// TIA Portal project "电厂_干燥机_V14" (V14)

(* hardware
DEVICE "S7-1200 station_1"  S7-1200 Station
   slot 0: "Rack_0"  Rack  V1.0
   slot 1: "PLC_1"  CPU 1214C AC/DC/Rly  6ES7 214-1BG40-0XB0  V4.2
   slot 101: "CM 1242-5"  CM 1242-5  6GK7 242-5DX30-0XE0  V1.0
DEVICE "HMI_2"  KTP700 Basic PN
   slot 0: "KTP700 Basic PN"  KTP700 Basic PN  6AV2 123-2GB03-0AX0  14.0.0.0
   slot 1: "HMI_RT_2"  KTP700 Basic PN  6AV2 123-2GB03-0AX0  14.0.0.0
   slot 5: "HMI_2.IE_CP_1"  PROFINET Interface  14.0.0.0
      slot 1: "PROFINET Interface_1"  PROFINET Interface
         slot 1: "Port_1"  Port
*)

// ===== PLC "PLC_1"  CPU 1214C AC/DC/Rly =====

VAR_GLOBAL   // PLC tag table "默认变量表"
   "System_Byte" AT %MB1 : Byte;
   "FirstScan" AT %M1.0 : Bool;
   "DiagStatusUpdate" AT %M1.1 : Bool;
   "AlwaysTRUE" AT %M1.2 : Bool;
   "AlwaysFALSE" AT %M1.3 : Bool;
   "Clock_Byte" AT %MB0 : Byte;
   "BClock_10Hz" AT %M0.0 : Bool;
   "Clock_5Hz" AT %M0.1 : Bool;
   "Clock_2.5Hz" AT %M0.2 : Bool;
   "Clock_2Hz" AT %M0.3 : Bool;
   "Clock_1.25Hz" AT %M0.4 : Bool;
   "Clock_1Hz" AT %M0.5 : Bool;
   "Clock_0.625Hz" AT %M0.6 : Bool;
   "Clock_0.5Hz" AT %M0.7 : Bool;
   "MB_COMM_LOAD_DONE" AT %M1.4 : Bool;
   "MB_COMM_LOAD_ERROR" AT %M1.5 : Bool;
   "MB_COMM_LOAD_STATUS" AT %MW1 : UInt;
   "MB_SLAVE_EN" AT %M1.6 : Bool;
END_VAR

VAR_GLOBAL   // PLC tag table "IO"
   "露点温度" AT %IW64 : Int;
   "加热温度" AT %IW66 : Int;
   "开机" AT %I0.0 : Bool;
   "停机" AT %I0.1 : Bool;
   "本地远程转换" AT %I0.2 : Bool;
   "远程开机" AT %I0.3 : Bool;
   "远程停机" AT %I0.4 : Bool;
   "进气低压" AT %I0.6 : Bool;
   "A塔进气阀" AT %Q0.0 : Bool;
   "B塔进气阀" AT %Q0.1 : Bool;
   "A塔排气阀" AT %Q0.2 : Bool;
   "B塔排气阀" AT %Q0.3 : Bool;
   "主加热" AT %Q0.4 : Bool;
   "辅加热" AT %Q0.5 : Bool;
   "运行指示" AT %Q0.6 : Bool;
   "故障指示" AT %Q0.7 : Bool;
   "远程指示" AT %Q1.0 : Bool;
END_VAR

// folder: IO

DATA_BLOCK "AI_conversion_DB"   // DB5
{ S7_Optimized_Access := 'TRUE' }
VERSION : 0.1
// stored: InstanceOfName ai_conversion
"ai_conversion"
BEGIN
END_DATA_BLOCK

// folder: Logic

DATA_BLOCK "PARAM_CONFIG_DB"   // DB6
{ S7_Optimized_Access := 'TRUE' }
VERSION : 0.1
// stored: InstanceOfName PARAM_Config
"PARAM_Config"
BEGIN
END_DATA_BLOCK

DATA_BLOCK "CTR_CYCLIC_DB"   // DB7
{ S7_Optimized_Access := 'TRUE' }
VERSION : 0.1
// stored: InstanceOfName CTR_Cyclic
"CTR_Cyclic"
BEGIN
END_DATA_BLOCK

DATA_BLOCK "AlarmError_DB"   // DB8
{ S7_Optimized_Access := 'TRUE' }
VERSION : 0.1
// stored: InstanceOfName Alarm_Error
"Alarm_Error"
BEGIN
END_DATA_BLOCK

// folder: ModbusRTU

DATA_BLOCK "mb_hold_reg"   // DB3
{ S7_Optimized_Access := 'FALSE' }
VERSION : 0.1
   VAR
      hold_registers : Array[0..99] of UInt;
   END_VAR
BEGIN
END_DATA_BLOCK

DATA_BLOCK "modbusrtu_DB"   // DB4
{ S7_Optimized_Access := 'TRUE' }
VERSION : 0.1
// stored: InstanceOfName modbusrtu
"modbusrtu"
BEGIN
END_DATA_BLOCK

// folder: (top level)

ORGANIZATION_BLOCK "Main"   // OB1, LAD, ProgramCycle
TITLE = "Main Program Sweep (Cycle)"
{ S7_Optimized_Access := 'TRUE' }
VERSION : 0.1
   VAR_TEMP   // added for the SCL form of the ladder/FBD networks
      _w1 : Bool;
   END_VAR
BEGIN

REGION Network 1: PARAM_Config
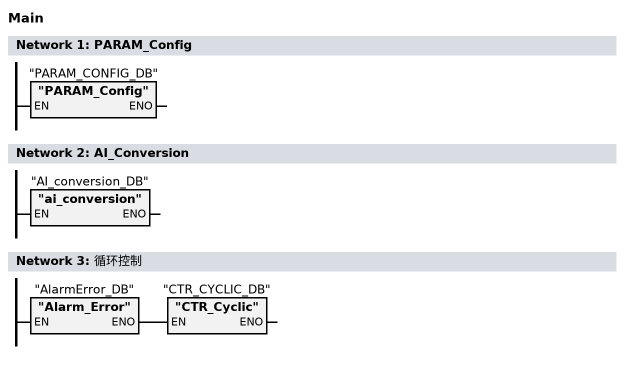
   RUNG wire#powerrail
      "PARAM_CONFIG_DB"()
   END_RUNG
   // the same network as SCL:
   "PARAM_CONFIG_DB"();   // "PARAM_Config"
END_REGION

REGION Network 2: AI_Conversion
   RUNG wire#powerrail
      "AI_conversion_DB"()
   END_RUNG
   // the same network as SCL:
   "AI_conversion_DB"();   // "ai_conversion"
END_REGION

REGION Network 3: 循环控制
   RUNG wire#powerrail
      "AlarmError_DB"()
      "CTR_CYCLIC_DB"()
   END_RUNG
   // the same network as SCL:
   "AlarmError_DB"(ENO => #_w1);   // "Alarm_Error"
   IF #_w1 THEN
       "CTR_CYCLIC_DB"();   // "CTR_Cyclic"
   END_IF;
END_REGION
END_ORGANIZATION_BLOCK

ORGANIZATION_BLOCK "Startup"   // OB100, LAD, Startup
TITLE = "Complete Restart"
{ S7_Optimized_Access := 'TRUE' }
VERSION : 0.1
   VAR_INPUT
      LostRetentive : Bool;   // True if retentive data are lost
      LostRTC : Bool;   // True if date and time are lost
   END_VAR
BEGIN

REGION Network 1: 运行时间计时初始化
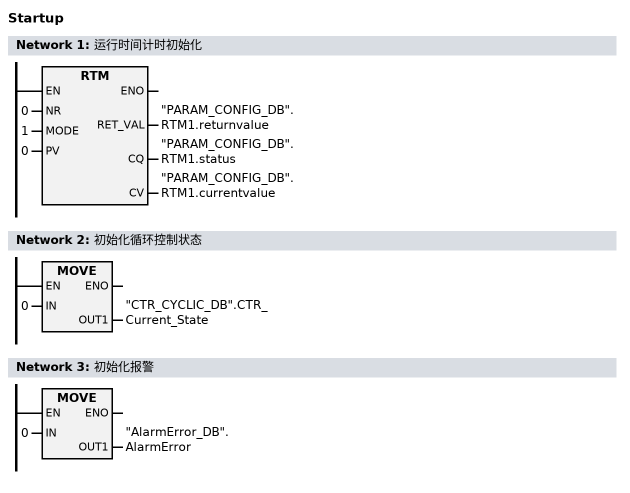
   "PARAM_CONFIG_DB".RTM1.returnvalue := RTM(NR := 0,
                           MODE := 1,
                           PV := 0,
                           CQ => "PARAM_CONFIG_DB".RTM1.status,
                           CV => "PARAM_CONFIG_DB".RTM1.currentvalue);
END_REGION

REGION Network 2: 初始化循环控制状态
   RUNG wire#powerrail
      Move(in := 0, out1 => "CTR_CYCLIC_DB".CTR_Current_State)
   END_RUNG
   // the same network as SCL:
   "CTR_CYCLIC_DB".CTR_Current_State := 0;
END_REGION

REGION Network 3: 初始化报警
   RUNG wire#powerrail
      Move(in := 0, out1 => "AlarmError_DB".AlarmError)
   END_RUNG
   // the same network as SCL:
   "AlarmError_DB".AlarmError := 0;
END_REGION
END_ORGANIZATION_BLOCK

// folder: IO

FUNCTION_BLOCK "ai_conversion"   // FB2, LAD
{ S7_Optimized_Access := 'TRUE' }
VERSION : 0.1
   VAR
      露点温度ac : Real;
      加热温度ac : Real;
   END_VAR
BEGIN

REGION Network 1: 露点温度线性变换
   // 露点温度传感器范围:-80-20摄氏度
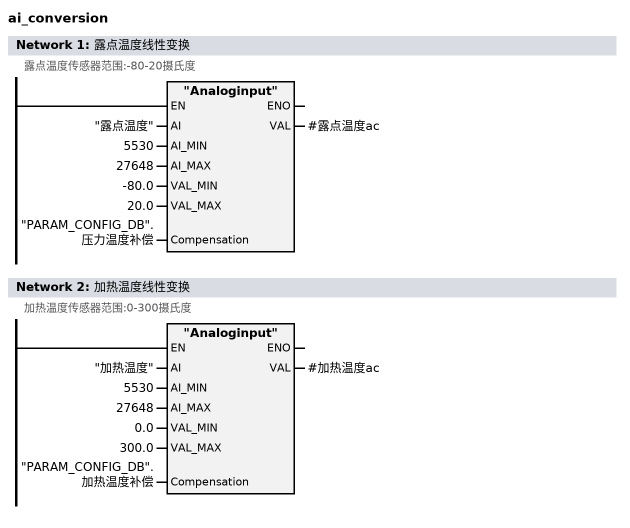
   RUNG wire#powerrail
      "Analoginput"(AI := "露点温度", AI_MIN := 5530, AI_MAX := 27648, VAL_MIN := -80.0, VAL_MAX := 20.0, Compensation := "PARAM_CONFIG_DB".压力温度补偿, VAL => #露点温度ac)
   END_RUNG
   // the same network as SCL:
   "Analoginput"(AI := "露点温度",
                 AI_MIN := 5530,
                 AI_MAX := 27648,
                 VAL_MIN := -80.0,
                 VAL_MAX := 20.0,
                 Compensation := "PARAM_CONFIG_DB".压力温度补偿,
                 VAL => #露点温度ac);
END_REGION

REGION Network 2: 加热温度线性变换
   // 加热温度传感器范围:0-300摄氏度
   RUNG wire#powerrail
      "Analoginput"(AI := "加热温度", AI_MIN := 5530, AI_MAX := 27648, VAL_MIN := 0.0, VAL_MAX := 300.0, Compensation := "PARAM_CONFIG_DB".加热温度补偿, VAL => #加热温度ac)
   END_RUNG
   // the same network as SCL:
   "Analoginput"(AI := "加热温度",
                 AI_MIN := 5530,
                 AI_MAX := 27648,
                 VAL_MIN := 0.0,
                 VAL_MAX := 300.0,
                 Compensation := "PARAM_CONFIG_DB".加热温度补偿,
                 VAL => #加热温度ac);
END_REGION
END_FUNCTION_BLOCK

FUNCTION "Analoginput" : Void   // FC71, LAD
TITLE = 模拟输入量处理
{ S7_Optimized_Access := 'TRUE' }
VERSION : 0.1
   VAR_INPUT
      AI : Int;   // 待处理模拟量
      AI_MIN : Int;   // 模拟量下限值
      AI_MAX : Int;   // 模拟量上限值
      VAL_MIN : Real;   // 实际值下限值
      VAL_MAX : Real;   // 实际值上限值
      Compensation : Real;
   END_VAR
   VAR_OUTPUT
      VAL : Real;   // 转换后的值
   END_VAR
   VAR_TEMP
      NORM_Out : Real;   // 模拟标准量
      SCALE_Out : Real;
   END_VAR
BEGIN

REGION Network 1: 标准化和缩放输入模拟量
   // 如果输入大于0,进行线性变换,否则赋值为0. / 输入模拟量是负值时,置零;
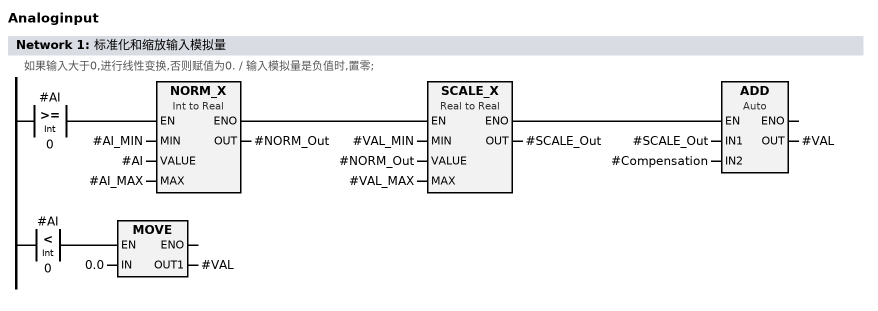
   RUNG wire#powerrail
      { S7_Templates := "SrcType := Int" } GE_Contact(in1 := #AI, in2 := 0)
      { S7_Templates := "[SrcType := Int, DestType := Real]"; S7_GenerateENO := "TRUE" } Normalize(min := #AI_MIN, value := #AI, max := #AI_MAX, out => #NORM_Out)
      { S7_Templates := "[SrcType := Real, DestType := Real]"; S7_GenerateENO := "TRUE" } Scale(min := #VAL_MIN, value := #NORM_Out, max := #VAL_MAX, out => #SCALE_Out)
      Add(in1 := #SCALE_Out, in2 := #Compensation, out => #VAL)
   END_RUNG
   RUNG wire#powerrail
      { S7_Templates := "SrcType := Int" } LT_Contact(in1 := #AI, in2 := 0)
      { S7_GenerateENO := "TRUE" } Move(in := 0.0, out1 => #VAL)
   END_RUNG
   // the same network as SCL:
   // ENO of a box is taken as its EN; it also drops when the box reports an error
   IF #AI >= 0 THEN
       #NORM_Out := NORM_X(MIN := #AI_MIN, VALUE := #AI, MAX := #AI_MAX);
       #SCALE_Out := SCALE_X(MIN := #VAL_MIN, VALUE := #NORM_Out, MAX := #VAL_MAX);
       #VAL := #SCALE_Out + #Compensation;
   END_IF;
   IF #AI < 0 THEN #VAL := 0.0; END_IF;
END_REGION
END_FUNCTION

// folder: Logic

FUNCTION_BLOCK "PARAM_Config"   // FB3, LAD
{ S7_Optimized_Access := 'TRUE' }
VERSION : 0.1
   VAR RETAIN
      主加热温度上限 : UInt := 120;   // 0～300℃
      主加热温度下限 : UInt := 100;   // 0～300℃
      加热超限温度报警 : UInt := 180;   // 0～300℃
      露点超限温度 : Int := -10;   // -500℃～500℃
      加热温度补偿 : Int := 0;   // -500℃～500℃
      压力温度补偿 : Int := 0;   // -500℃～500℃
      工作露点设定 : Int := -30;   // -500℃～500℃
      停机充压时间 : UDInt := 60;   // 3～999秒
      A塔工作B塔待再生 : UDInt := 10;   // 0～3600秒
      A塔工作B塔热再生 : UDInt := 25;   // 0～3600分
      A塔工作B塔吹冷 : UDInt := 15;   // 0～3600分
      A塔工作B塔充压 : UDInt := 8;   // 0～3600分
      A塔B塔均压 : UDInt := 10;   // 0～3600秒
      故障判断延时 : UInt := 5;   // 0～3600秒
      保养时间设定 : UDInt := 0;   // 0～100000h
      从站地址 : UInt := 2;   // 1～255
      露点控制最长延时 : UInt := 60;   // 0～3600分
   END_VAR
   VAR
      BT_Function : Struct
         BT_Runtime_Reset : Bool;
         BT_RuntimeReset_PREStatus : Bool;
      END_STRUCT;
      IEC_Timer_0_Instance : TONR_TIME;
      RTM1 : Struct
         returnvalue : Int;
         status : Bool;
         currentvalue : DInt;
         mode : UInt;
      END_STRUCT;
      MaintainTime_CountdownValue : Real;
   END_VAR
   VAR CONSTANT
      主加热温度上限_default : UInt := 120;   // default
      主加热温度下限_default : UInt := 100;   // default
      加热超限温度报警_default : UInt := 180;   // default
      露点超限温度_default : Int := -10;   // default
      加热温度补偿_default : Int := 0;   // default
      露点温度补偿_default : Int := 0;   // default
      工作露点设定_default : Int := -30;   // default
      停机充压时间_default : UInt := 30;   // default
      A塔工作B塔待再生_default : UInt := 10;   // default
      A塔工作B塔热再生_default : UInt := 25;   // default
      A塔工作B塔吹冷_default : UInt := 15;   // default
      A塔工作B塔充压_default : UInt := 8;   // default
      A塔B塔均压_default : UInt := 10;   // default
      故障判断延时_default : UInt := 5;   // default
      保养时间设定_default : UDInt := 0;   // default
      从站地址_default : UInt := 2;   // default
      露点控制最长延时_default : UInt := 60;   // default
   END_VAR
   VAR_TEMP   // added for the SCL form of the ladder/FBD networks
      _w1 : Bool;
   END_VAR
BEGIN

REGION Network 1: 运行时间复位
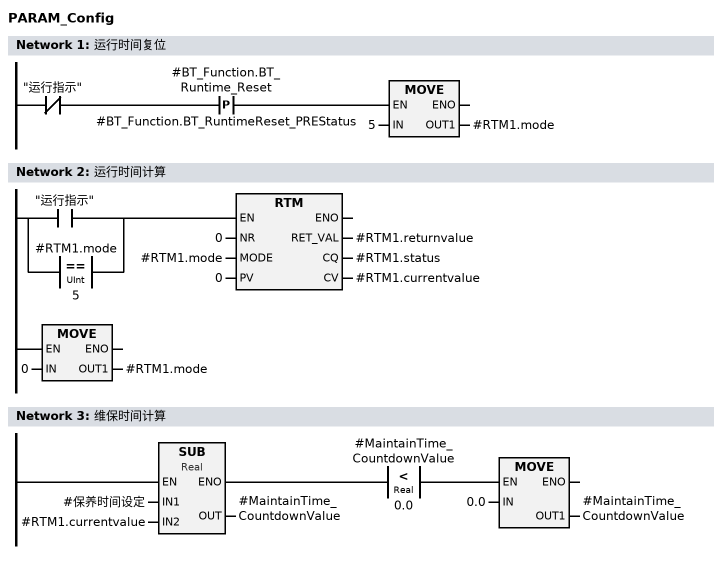
   RUNG wire#powerrail
      I_Contact( "运行指示" )
      P_Contact(operand := #BT_Function.BT_Runtime_Reset, bit := #BT_Function.BT_RuntimeReset_PREStatus)
      Move(in := 5, out1 => #RTM1.mode)
   END_RUNG
   // the same network as SCL:
   #_w1 := NOT "运行指示" AND #BT_Function.BT_Runtime_Reset AND NOT #BT_Function.BT_RuntimeReset_PREStatus;   // rising edge of #BT_Function.BT_Runtime_Reset
   #BT_Function.BT_RuntimeReset_PREStatus := #BT_Function.BT_Runtime_Reset;
   IF #_w1 THEN #RTM1.mode := 5; END_IF;
END_REGION

REGION Network 2: 运行时间计算
   IF "运行指示" OR (#RTM1.mode = 5) THEN
       #RTM1.returnvalue := RTM(NR := 0, MODE := #RTM1.mode, PV := 0, CQ => #RTM1.status, CV => #RTM1.currentvalue);
   END_IF;
   #RTM1.mode := 0;
END_REGION

REGION Network 3: 维保时间计算
   RUNG wire#powerrail
      { S7_Templates := "SrcType := Real" } Sub(in1 := #保养时间设定, in2 := #RTM1.currentvalue, out => #MaintainTime_CountdownValue)
      { S7_Templates := "SrcType := Real" } LT_Contact(in1 := #MaintainTime_CountdownValue, in2 := 0.0)
      Move(in := 0.0, out1 => #MaintainTime_CountdownValue)
   END_RUNG
   // the same network as SCL:
   #MaintainTime_CountdownValue := #保养时间设定 - #RTM1.currentvalue;
   IF #MaintainTime_CountdownValue < 0.0 THEN #MaintainTime_CountdownValue := 0.0; END_IF;
END_REGION
END_FUNCTION_BLOCK

FUNCTION_BLOCK "CTR_Cyclic"   // FB4, LAD
{ S7_Optimized_Access := 'TRUE' }
VERSION : 0.1
   VAR
      CTR_Current_State : UInt;   // 当前控制循环的步骤
      Total_Error : Bool;
      IEC_Timer_0_Instance : TON_TIME;
      Cyclic_Switch_Flag : Bool;
      BT_function : Struct
         BT_Atower_Open : Bool;
         BT_Atower_Open_PRE : Bool;
         BT_Btower_Open : Bool;
         BT_Btower_Open_PRE : Bool;
         BT_Stop : Bool;
         BT_Stop_PRE : Bool;
      END_STRUCT;
      BT_LocalRemoteSwitch : Bool;
   END_VAR
   VAR RETAIN
      BT_TimeCTRL_DCTR_Switch : Bool;
   END_VAR
   VAR
      RemoteStart_PRE : Bool;
      RemoteStop_PRE : Bool;
      JXStart_PRE : Bool;
      JXStop_PRE : Bool;
      IEC_Timer_0_Instance1 : TON_TIME;
      IEC_Timer_0_Instance2 : TON_TIME;
      IEC_Timer_0_Instance3 : TON_TIME;
      IEC_Timer_0_Instance4 : TON_TIME;
      IEC_Timer_0_Instance5 : TON_TIME;
      IEC_Timer_0_Instance6 : TON_TIME;
      IEC_Timer_0_Instance7 : TON_TIME;
      IEC_Timer_0_Instance8 : TON_TIME;
      IEC_Timer_0_Instance9 : TON_TIME;
      IEC_Timer_0_Instance10 : TON_TIME;
      IEC_Timer_0_Instance11 : TON_TIME;
      IEC_Timer_0_Instance5_1 : TON_TIME;
      IEC_Timer_0_Instance10_1 : TON_TIME;
      Count_Down_Time : UDInt;
   END_VAR
   VAR_TEMP
      A塔工作B塔待再生_Interval : Time;
      A塔工作B塔热热再生_Interval : Time;
      A塔工作B塔热再生_Interval : Time;
      A塔工作B塔吹冷_Interval : Time;
      A塔工作B塔充压_Interval : Time;
      A塔B塔均压_Interval : Time;
      B塔工作A塔待再生_Interval : Time;
      B塔工作A塔热再生_Interval : Time;
      B塔工作A塔吹冷_Interval : Time;
      B塔工作A塔充压_Interval : Time;
      B塔A塔均压_Interval : Time;
      停机充压时间_Interval : Time;
      A塔工作B塔待再生_Interval_1 : UDInt;
      A塔工作B塔热热再生_Interval_1 : UDInt;
      A塔工作B塔热再生_Interval_1 : UDInt;
      A塔工作B塔吹冷_Interval_1 : UDInt;
      A塔工作B塔充压_Interval_1 : UDInt;
      A塔B塔均压_Interval_1 : UDInt;
      B塔工作A塔待再生_Interval_1 : UDInt;
      B塔工作A塔热再生_Interval_1 : UDInt;
      B塔工作A塔吹冷_Interval_1 : UDInt;
      B塔工作A塔充压_Interval_1 : UDInt;
      B塔A塔均压_Interval_1 : UDInt;
      停机充压时间_Interval_1 : UDInt;
      露点控制最长延时_Interval : Time;
      露点控制最长延时_Interval_1 : UDInt;
   END_VAR
   VAR_TEMP   // added for the SCL form of the ladder/FBD networks
      _w1 : Bool;
      _w2 : Bool;
      _w3 : Bool;
   END_VAR
BEGIN

REGION Network 1: Cyclic Switch
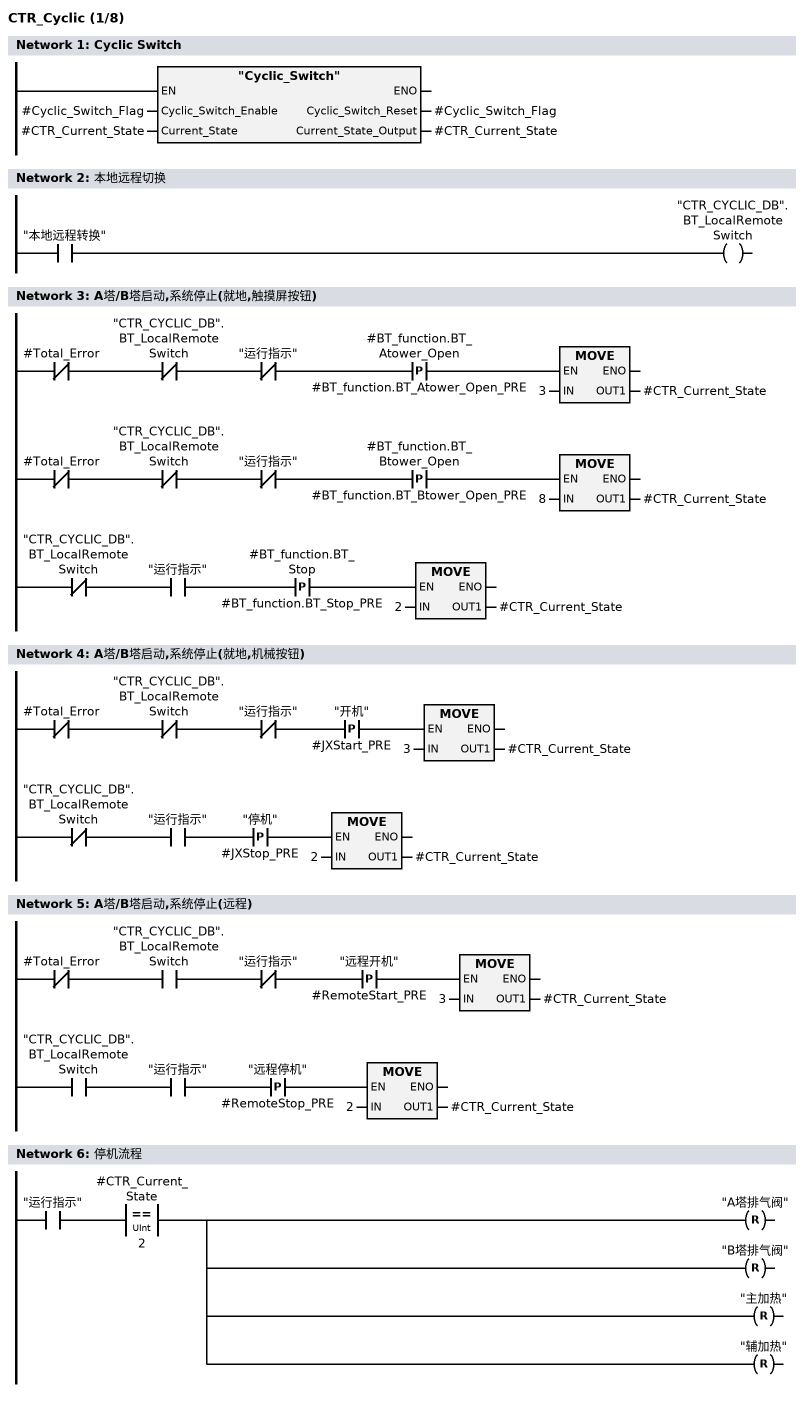
   RUNG wire#powerrail
      "Cyclic_Switch"(Cyclic_Switch_Enable := #Cyclic_Switch_Flag, Current_State := #CTR_Current_State, Cyclic_Switch_Reset => #Cyclic_Switch_Flag, Current_State_Output => #CTR_Current_State)
   END_RUNG
   // the same network as SCL:
   "Cyclic_Switch"(Cyclic_Switch_Enable := #Cyclic_Switch_Flag,
                   Current_State := #CTR_Current_State,
                   Cyclic_Switch_Reset => #Cyclic_Switch_Flag,
                   Current_State_Output => #CTR_Current_State);
END_REGION

REGION Network 2: 本地远程切换
   RUNG wire#powerrail
      Contact( "本地远程转换" )
      Coil( "CTR_CYCLIC_DB".BT_LocalRemoteSwitch )
   END_RUNG
   // the same network as SCL:
   "CTR_CYCLIC_DB".BT_LocalRemoteSwitch := "本地远程转换";
END_REGION

REGION Network 3: A塔/B塔启动,系统停止(就地,触摸屏按钮)
   RUNG wire#powerrail
      I_Contact( #Total_Error )
      I_Contact( "CTR_CYCLIC_DB".BT_LocalRemoteSwitch )
      I_Contact( "运行指示" )
      P_Contact(operand := #BT_function.BT_Atower_Open, bit := #BT_function.BT_Atower_Open_PRE)
      Move(in := 3, out1 => #CTR_Current_State)
   END_RUNG
   RUNG wire#powerrail
      I_Contact( #Total_Error )
      I_Contact( "CTR_CYCLIC_DB".BT_LocalRemoteSwitch )
      I_Contact( "运行指示" )
      P_Contact(operand := #BT_function.BT_Btower_Open, bit := #BT_function.BT_Btower_Open_PRE)
      Move(in := 8, out1 => #CTR_Current_State)
   END_RUNG
   RUNG wire#powerrail
      I_Contact( "CTR_CYCLIC_DB".BT_LocalRemoteSwitch )
      Contact( "运行指示" )
      P_Contact(operand := #BT_function.BT_Stop, bit := #BT_function.BT_Stop_PRE)
      Move(in := 2, out1 => #CTR_Current_State)
   END_RUNG
   // the same network as SCL:
   #_w1 := NOT #Total_Error AND NOT "CTR_CYCLIC_DB".BT_LocalRemoteSwitch AND NOT "运行指示" AND #BT_function.BT_Atower_Open AND NOT #BT_function.BT_Atower_Open_PRE;   // rising edge of #BT_function.BT_Atower_Open
   #BT_function.BT_Atower_Open_PRE := #BT_function.BT_Atower_Open;
   IF #_w1 THEN #CTR_Current_State := 3; END_IF;
   #_w2 := NOT #Total_Error AND NOT "CTR_CYCLIC_DB".BT_LocalRemoteSwitch AND NOT "运行指示" AND #BT_function.BT_Btower_Open AND NOT #BT_function.BT_Btower_Open_PRE;   // rising edge of #BT_function.BT_Btower_Open
   #BT_function.BT_Btower_Open_PRE := #BT_function.BT_Btower_Open;
   IF #_w2 THEN #CTR_Current_State := 8; END_IF;
   #_w3 := NOT "CTR_CYCLIC_DB".BT_LocalRemoteSwitch AND "运行指示" AND #BT_function.BT_Stop AND NOT #BT_function.BT_Stop_PRE;   // rising edge of #BT_function.BT_Stop
   #BT_function.BT_Stop_PRE := #BT_function.BT_Stop;
   IF #_w3 THEN #CTR_Current_State := 2; END_IF;
END_REGION

REGION Network 4: A塔/B塔启动,系统停止(就地,机械按钮)
   RUNG wire#powerrail
      I_Contact( #Total_Error )
      I_Contact( "CTR_CYCLIC_DB".BT_LocalRemoteSwitch )
      I_Contact( "运行指示" )
      P_Contact(operand := "开机", bit := #JXStart_PRE)
      Move(in := 3, out1 => #CTR_Current_State)
   END_RUNG
   RUNG wire#powerrail
      I_Contact( "CTR_CYCLIC_DB".BT_LocalRemoteSwitch )
      Contact( "运行指示" )
      P_Contact(operand := "停机", bit := #JXStop_PRE)
      Move(in := 2, out1 => #CTR_Current_State)
   END_RUNG
   // the same network as SCL:
   #_w1 := NOT #Total_Error AND NOT "CTR_CYCLIC_DB".BT_LocalRemoteSwitch AND NOT "运行指示" AND "开机" AND NOT #JXStart_PRE;   // rising edge of "开机"
   #JXStart_PRE := "开机";
   IF #_w1 THEN #CTR_Current_State := 3; END_IF;
   #_w2 := NOT "CTR_CYCLIC_DB".BT_LocalRemoteSwitch AND "运行指示" AND "停机" AND NOT #JXStop_PRE;   // rising edge of "停机"
   #JXStop_PRE := "停机";
   IF #_w2 THEN #CTR_Current_State := 2; END_IF;
END_REGION

REGION Network 5: A塔/B塔启动,系统停止(远程)
   RUNG wire#powerrail
      I_Contact( #Total_Error )
      Contact( "CTR_CYCLIC_DB".BT_LocalRemoteSwitch )
      I_Contact( "运行指示" )
      P_Contact(operand := "远程开机", bit := #RemoteStart_PRE)
      Move(in := 3, out1 => #CTR_Current_State)
   END_RUNG
   RUNG wire#powerrail
      Contact( "CTR_CYCLIC_DB".BT_LocalRemoteSwitch )
      Contact( "运行指示" )
      P_Contact(operand := "远程停机", bit := #RemoteStop_PRE)
      Move(in := 2, out1 => #CTR_Current_State)
   END_RUNG
   // the same network as SCL:
   #_w1 := NOT #Total_Error AND "CTR_CYCLIC_DB".BT_LocalRemoteSwitch AND NOT "运行指示" AND "远程开机" AND NOT #RemoteStart_PRE;   // rising edge of "远程开机"
   #RemoteStart_PRE := "远程开机";
   IF #_w1 THEN #CTR_Current_State := 3; END_IF;
   #_w2 := "CTR_CYCLIC_DB".BT_LocalRemoteSwitch AND "运行指示" AND "远程停机" AND NOT #RemoteStop_PRE;   // rising edge of "远程停机"
   #RemoteStop_PRE := "远程停机";
   IF #_w2 THEN #CTR_Current_State := 2; END_IF;
END_REGION

REGION Network 6: 停机流程
   RUNG wire#powerrail
      Contact( "运行指示" )
      { S7_Templates := "SrcType := UInt" } EQ_Contact(in1 := #CTR_Current_State, in2 := 2)
      wire#w1
      R_Coil( "A塔排气阀" )
   END_RUNG
   RUNG wire#w1
      R_Coil( "B塔排气阀" )
   END_RUNG
   RUNG wire#w1
      R_Coil( "主加热" )
   END_RUNG
   RUNG wire#w1
      R_Coil( "辅加热" )
   END_RUNG
   // the same network as SCL:
   IF "运行指示" AND (#CTR_Current_State = 2) THEN
       "A塔排气阀" := FALSE;
       "B塔排气阀" := FALSE;
       "主加热" := FALSE;
       "辅加热" := FALSE;
   END_IF;
END_REGION

REGION Network 7
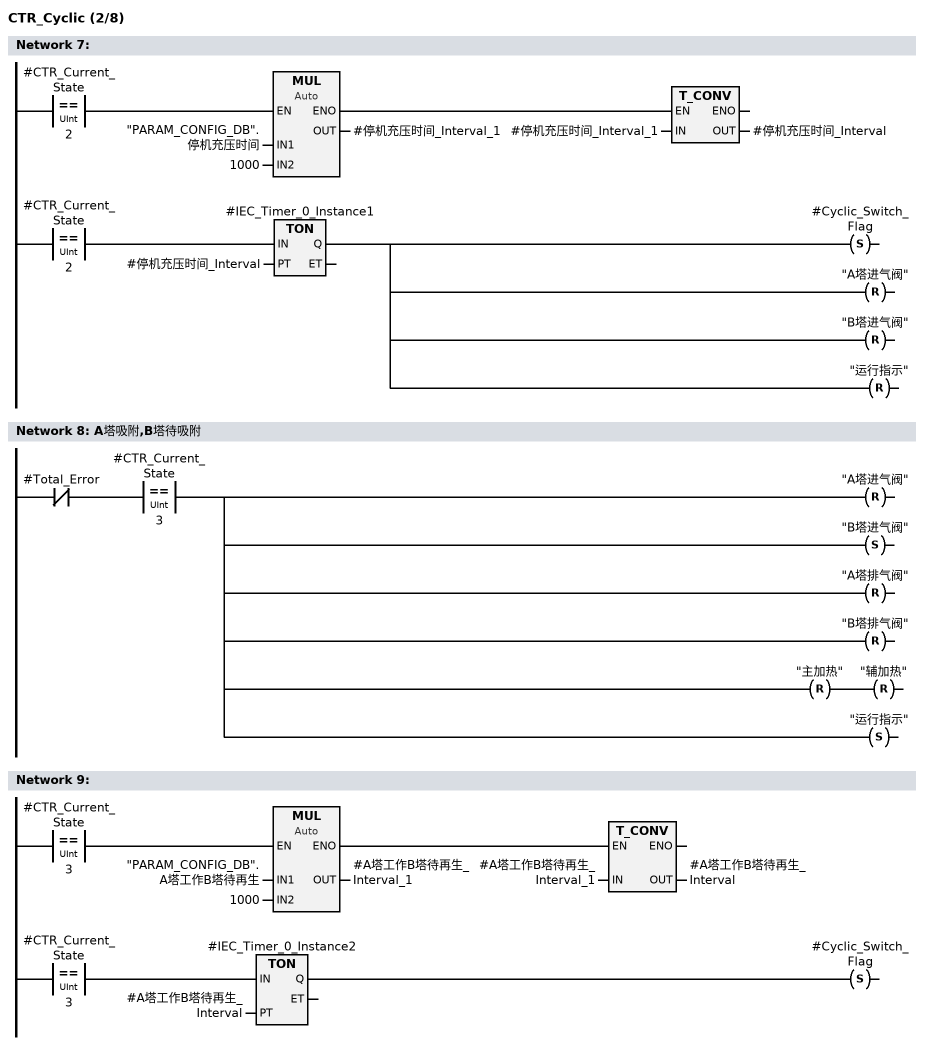
   IF #CTR_Current_State = 2 THEN
       #停机充压时间_Interval_1 := "PARAM_CONFIG_DB".停机充压时间 * 1000;
       #停机充压时间_Interval := T_CONV(IN := #停机充压时间_Interval_1);
   END_IF;
   #IEC_Timer_0_Instance1(IN := #CTR_Current_State = 2, PT := #停机充压时间_Interval);   // TON
   IF #IEC_Timer_0_Instance1.Q THEN
       #Cyclic_Switch_Flag := TRUE;
       "A塔进气阀" := FALSE;
       "B塔进气阀" := FALSE;
       "运行指示" := FALSE;
   END_IF;
END_REGION

REGION Network 8: A塔吸附,B塔待吸附
   RUNG wire#powerrail
      I_Contact( #Total_Error )
      { S7_Templates := "SrcType := UInt" } EQ_Contact(in1 := #CTR_Current_State, in2 := 3)
      wire#w1
      R_Coil( "A塔进气阀" )
   END_RUNG
   RUNG wire#w1
      S_Coil( "B塔进气阀" )
   END_RUNG
   RUNG wire#w1
      R_Coil( "A塔排气阀" )
   END_RUNG
   RUNG wire#w1
      R_Coil( "B塔排气阀" )
   END_RUNG
   RUNG wire#w1
      R_Coil( "主加热" )
      R_Coil( "辅加热" )
   END_RUNG
   RUNG wire#w1
      S_Coil( "运行指示" )
   END_RUNG
   // the same network as SCL:
   IF NOT #Total_Error AND (#CTR_Current_State = 3) THEN
       "A塔进气阀" := FALSE;
       "B塔进气阀" := TRUE;
       "A塔排气阀" := FALSE;
       "B塔排气阀" := FALSE;
       "主加热" := FALSE;
       "辅加热" := FALSE;
       "运行指示" := TRUE;
   END_IF;
END_REGION

REGION Network 9
   IF #CTR_Current_State = 3 THEN
       #A塔工作B塔待再生_Interval_1 := "PARAM_CONFIG_DB".A塔工作B塔待再生 * 1000;
       #A塔工作B塔待再生_Interval := T_CONV(IN := #A塔工作B塔待再生_Interval_1);
   END_IF;
   #IEC_Timer_0_Instance2(IN := #CTR_Current_State = 3, PT := #A塔工作B塔待再生_Interval);   // TON
   IF #IEC_Timer_0_Instance2.Q THEN #Cyclic_Switch_Flag := TRUE; END_IF;
END_REGION

REGION Network 10: A塔吸附,B塔热再生(主加热根据温度判断开断;)
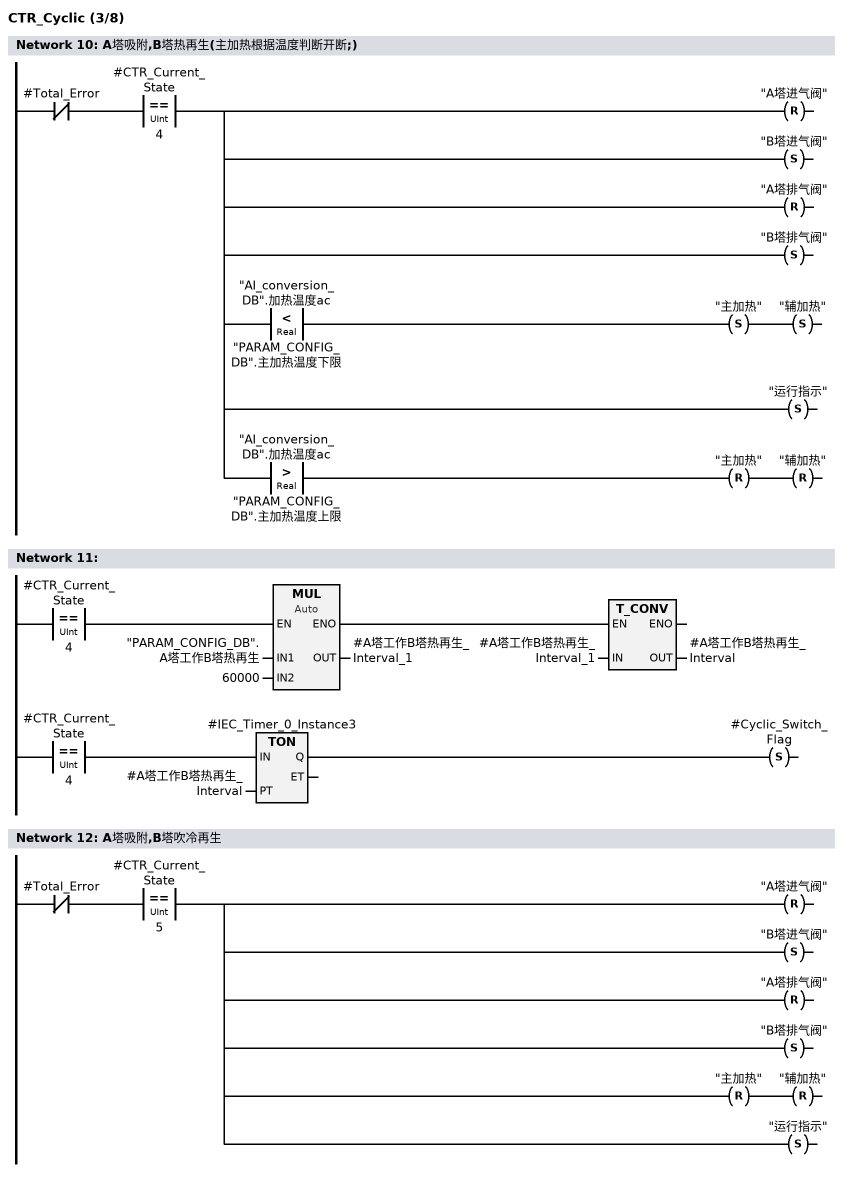
   RUNG wire#powerrail
      I_Contact( #Total_Error )
      { S7_Templates := "SrcType := UInt" } EQ_Contact(in1 := #CTR_Current_State, in2 := 4)
      wire#w1
      R_Coil( "A塔进气阀" )
   END_RUNG
   RUNG wire#w1
      S_Coil( "B塔进气阀" )
   END_RUNG
   RUNG wire#w1
      R_Coil( "A塔排气阀" )
   END_RUNG
   RUNG wire#w1
      S_Coil( "B塔排气阀" )
   END_RUNG
   RUNG wire#w1
      { S7_Templates := "SrcType := Real" } LT_Contact(in1 := "AI_conversion_DB".加热温度ac, in2 := "PARAM_CONFIG_DB".主加热温度下限)
      S_Coil( "主加热" )
      S_Coil( "辅加热" )
   END_RUNG
   RUNG wire#w1
      S_Coil( "运行指示" )
   END_RUNG
   RUNG wire#w1
      { S7_Templates := "SrcType := Real" } GT_Contact(in1 := "AI_conversion_DB".加热温度ac, in2 := "PARAM_CONFIG_DB".主加热温度上限)
      R_Coil( "主加热" )
      R_Coil( "辅加热" )
   END_RUNG
   // the same network as SCL:
   #_w1 := NOT #Total_Error AND (#CTR_Current_State = 4);
   IF #_w1 THEN
       "A塔进气阀" := FALSE;
       "B塔进气阀" := TRUE;
       "A塔排气阀" := FALSE;
       "B塔排气阀" := TRUE;
   END_IF;
   IF #_w1 AND ("AI_conversion_DB".加热温度ac < "PARAM_CONFIG_DB".主加热温度下限) THEN
       "主加热" := TRUE;
       "辅加热" := TRUE;
   END_IF;
   IF #_w1 THEN "运行指示" := TRUE; END_IF;
   IF #_w1 AND ("AI_conversion_DB".加热温度ac > "PARAM_CONFIG_DB".主加热温度上限) THEN
       "主加热" := FALSE;
       "辅加热" := FALSE;
   END_IF;
END_REGION

REGION Network 11
   IF #CTR_Current_State = 4 THEN
       #A塔工作B塔热再生_Interval_1 := "PARAM_CONFIG_DB".A塔工作B塔热再生 * 60000;
       #A塔工作B塔热再生_Interval := T_CONV(IN := #A塔工作B塔热再生_Interval_1);
   END_IF;
   #IEC_Timer_0_Instance3(IN := #CTR_Current_State = 4, PT := #A塔工作B塔热再生_Interval);   // TON
   IF #IEC_Timer_0_Instance3.Q THEN #Cyclic_Switch_Flag := TRUE; END_IF;
END_REGION

REGION Network 12: A塔吸附,B塔吹冷再生
   RUNG wire#powerrail
      I_Contact( #Total_Error )
      { S7_Templates := "SrcType := UInt" } EQ_Contact(in1 := #CTR_Current_State, in2 := 5)
      wire#w1
      R_Coil( "A塔进气阀" )
   END_RUNG
   RUNG wire#w1
      S_Coil( "B塔进气阀" )
   END_RUNG
   RUNG wire#w1
      R_Coil( "A塔排气阀" )
   END_RUNG
   RUNG wire#w1
      S_Coil( "B塔排气阀" )
   END_RUNG
   RUNG wire#w1
      R_Coil( "主加热" )
      R_Coil( "辅加热" )
   END_RUNG
   RUNG wire#w1
      S_Coil( "运行指示" )
   END_RUNG
   // the same network as SCL:
   IF NOT #Total_Error AND (#CTR_Current_State = 5) THEN
       "A塔进气阀" := FALSE;
       "B塔进气阀" := TRUE;
       "A塔排气阀" := FALSE;
       "B塔排气阀" := TRUE;
       "主加热" := FALSE;
       "辅加热" := FALSE;
       "运行指示" := TRUE;
   END_IF;
END_REGION

REGION Network 13
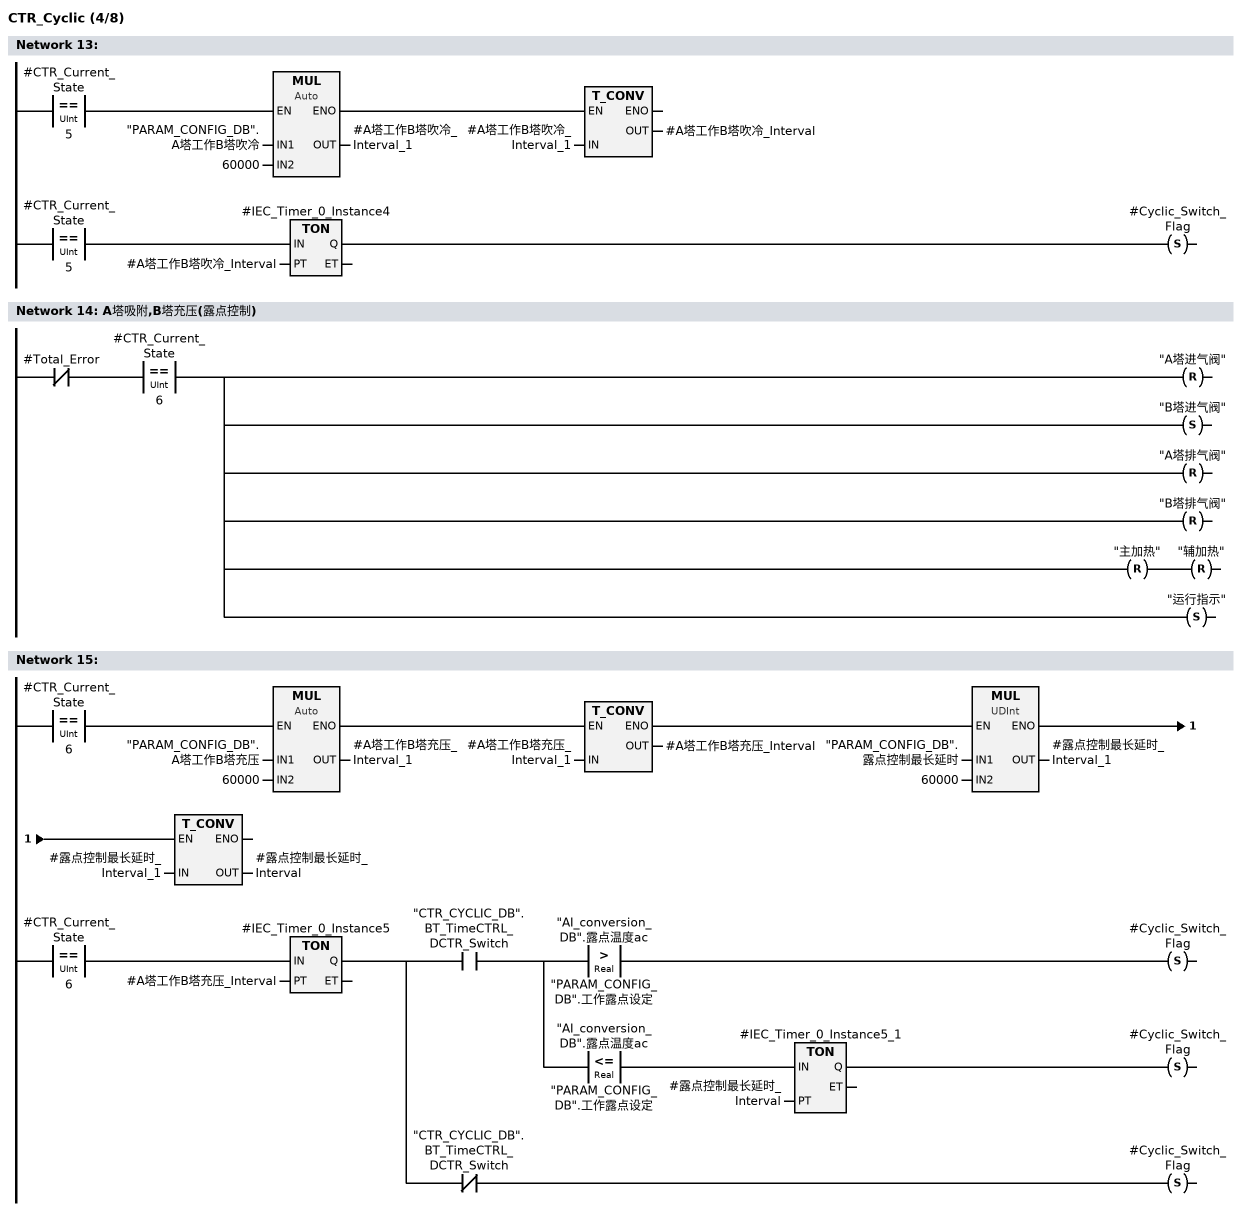
   IF #CTR_Current_State = 5 THEN
       #A塔工作B塔吹冷_Interval_1 := "PARAM_CONFIG_DB".A塔工作B塔吹冷 * 60000;
       #A塔工作B塔吹冷_Interval := T_CONV(IN := #A塔工作B塔吹冷_Interval_1);
   END_IF;
   #IEC_Timer_0_Instance4(IN := #CTR_Current_State = 5, PT := #A塔工作B塔吹冷_Interval);   // TON
   IF #IEC_Timer_0_Instance4.Q THEN #Cyclic_Switch_Flag := TRUE; END_IF;
END_REGION

REGION Network 14: A塔吸附,B塔充压(露点控制)
   RUNG wire#powerrail
      I_Contact( #Total_Error )
      { S7_Templates := "SrcType := UInt" } EQ_Contact(in1 := #CTR_Current_State, in2 := 6)
      wire#w1
      R_Coil( "A塔进气阀" )
   END_RUNG
   RUNG wire#w1
      S_Coil( "B塔进气阀" )
   END_RUNG
   RUNG wire#w1
      R_Coil( "A塔排气阀" )
   END_RUNG
   RUNG wire#w1
      R_Coil( "B塔排气阀" )
   END_RUNG
   RUNG wire#w1
      R_Coil( "主加热" )
      R_Coil( "辅加热" )
   END_RUNG
   RUNG wire#w1
      S_Coil( "运行指示" )
   END_RUNG
   // the same network as SCL:
   IF NOT #Total_Error AND (#CTR_Current_State = 6) THEN
       "A塔进气阀" := FALSE;
       "B塔进气阀" := TRUE;
       "A塔排气阀" := FALSE;
       "B塔排气阀" := FALSE;
       "主加热" := FALSE;
       "辅加热" := FALSE;
       "运行指示" := TRUE;
   END_IF;
END_REGION

REGION Network 15
   // ENO of a box is taken as its EN; it also drops when the box reports an error
   IF #CTR_Current_State = 6 THEN
       #A塔工作B塔充压_Interval_1 := "PARAM_CONFIG_DB".A塔工作B塔充压 * 60000;
       #A塔工作B塔充压_Interval := T_CONV(IN := #A塔工作B塔充压_Interval_1);
       #露点控制最长延时_Interval_1 := "PARAM_CONFIG_DB".露点控制最长延时 * 60000;
       #露点控制最长延时_Interval := T_CONV(IN := #露点控制最长延时_Interval_1);
   END_IF;
   #IEC_Timer_0_Instance5(IN := #CTR_Current_State = 6, PT := #A塔工作B塔充压_Interval);   // TON
   #_w1 := #IEC_Timer_0_Instance5.Q AND "CTR_CYCLIC_DB".BT_TimeCTRL_DCTR_Switch;
   IF #_w1 AND ("AI_conversion_DB".露点温度ac > "PARAM_CONFIG_DB".工作露点设定) THEN
       #Cyclic_Switch_Flag := TRUE;
   END_IF;
   #IEC_Timer_0_Instance5_1(IN := #_w1 AND ("AI_conversion_DB".露点温度ac <= "PARAM_CONFIG_DB".工作露点设定),   // TON
                           PT := #露点控制最长延时_Interval);
   IF #IEC_Timer_0_Instance5_1.Q THEN #Cyclic_Switch_Flag := TRUE; END_IF;
   IF #IEC_Timer_0_Instance5.Q AND NOT "CTR_CYCLIC_DB".BT_TimeCTRL_DCTR_Switch THEN
       #Cyclic_Switch_Flag := TRUE;
   END_IF;
END_REGION

REGION Network 16: A塔吸附,B塔均压
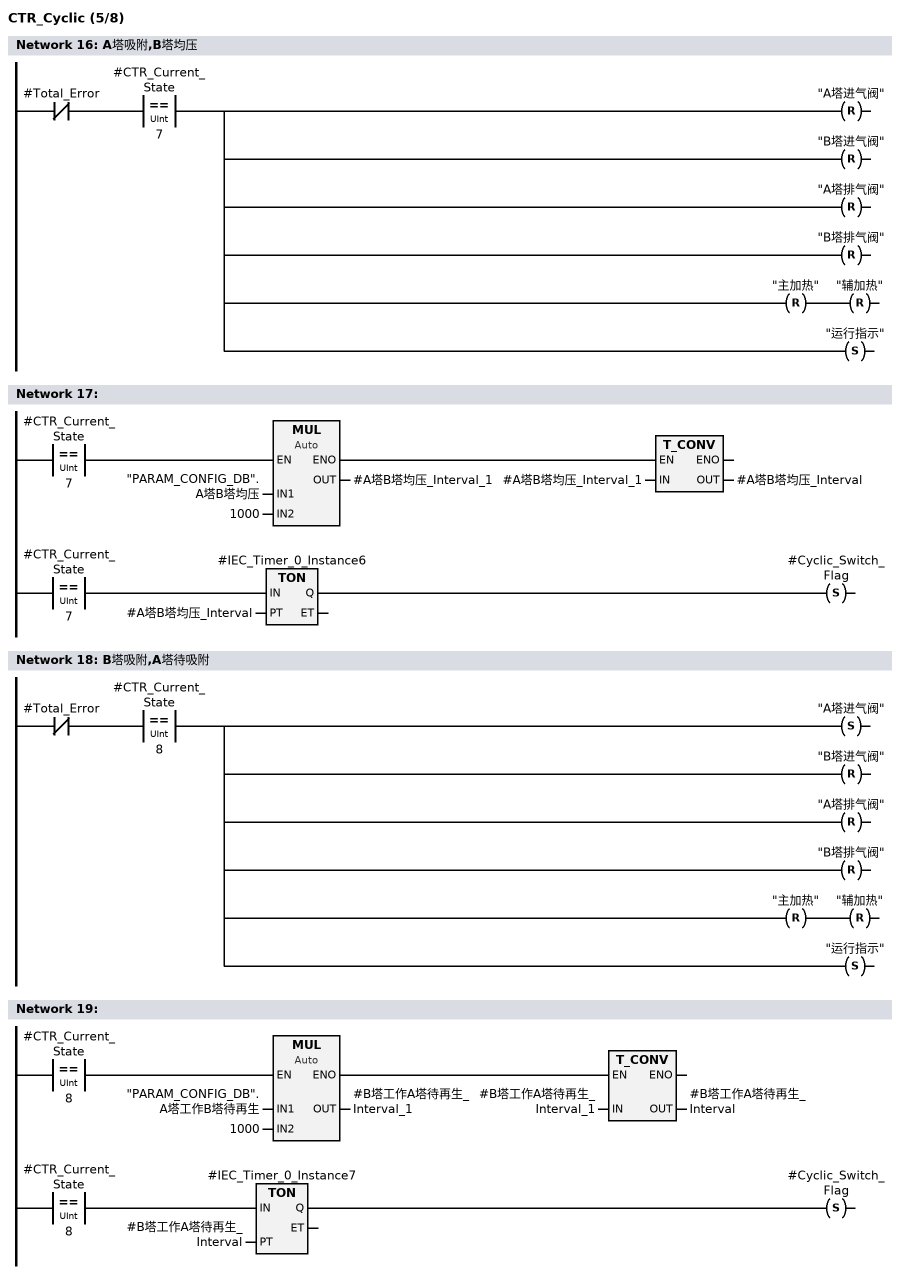
   RUNG wire#powerrail
      I_Contact( #Total_Error )
      { S7_Templates := "SrcType := UInt" } EQ_Contact(in1 := #CTR_Current_State, in2 := 7)
      wire#w1
      R_Coil( "A塔进气阀" )
   END_RUNG
   RUNG wire#w1
      R_Coil( "B塔进气阀" )
   END_RUNG
   RUNG wire#w1
      R_Coil( "A塔排气阀" )
   END_RUNG
   RUNG wire#w1
      R_Coil( "B塔排气阀" )
   END_RUNG
   RUNG wire#w1
      R_Coil( "主加热" )
      R_Coil( "辅加热" )
   END_RUNG
   RUNG wire#w1
      S_Coil( "运行指示" )
   END_RUNG
   // the same network as SCL:
   IF NOT #Total_Error AND (#CTR_Current_State = 7) THEN
       "A塔进气阀" := FALSE;
       "B塔进气阀" := FALSE;
       "A塔排气阀" := FALSE;
       "B塔排气阀" := FALSE;
       "主加热" := FALSE;
       "辅加热" := FALSE;
       "运行指示" := TRUE;
   END_IF;
END_REGION

REGION Network 17
   IF #CTR_Current_State = 7 THEN
       #A塔B塔均压_Interval_1 := "PARAM_CONFIG_DB".A塔B塔均压 * 1000;
       #A塔B塔均压_Interval := T_CONV(IN := #A塔B塔均压_Interval_1);
   END_IF;
   #IEC_Timer_0_Instance6(IN := #CTR_Current_State = 7, PT := #A塔B塔均压_Interval);   // TON
   IF #IEC_Timer_0_Instance6.Q THEN #Cyclic_Switch_Flag := TRUE; END_IF;
END_REGION

REGION Network 18: B塔吸附,A塔待吸附
   RUNG wire#powerrail
      I_Contact( #Total_Error )
      { S7_Templates := "SrcType := UInt" } EQ_Contact(in1 := #CTR_Current_State, in2 := 8)
      wire#w1
      S_Coil( "A塔进气阀" )
   END_RUNG
   RUNG wire#w1
      R_Coil( "B塔进气阀" )
   END_RUNG
   RUNG wire#w1
      R_Coil( "A塔排气阀" )
   END_RUNG
   RUNG wire#w1
      R_Coil( "B塔排气阀" )
   END_RUNG
   RUNG wire#w1
      R_Coil( "主加热" )
      R_Coil( "辅加热" )
   END_RUNG
   RUNG wire#w1
      S_Coil( "运行指示" )
   END_RUNG
   // the same network as SCL:
   IF NOT #Total_Error AND (#CTR_Current_State = 8) THEN
       "A塔进气阀" := TRUE;
       "B塔进气阀" := FALSE;
       "A塔排气阀" := FALSE;
       "B塔排气阀" := FALSE;
       "主加热" := FALSE;
       "辅加热" := FALSE;
       "运行指示" := TRUE;
   END_IF;
END_REGION

REGION Network 19
   IF #CTR_Current_State = 8 THEN
       #B塔工作A塔待再生_Interval_1 := "PARAM_CONFIG_DB".A塔工作B塔待再生 * 1000;
       #B塔工作A塔待再生_Interval := T_CONV(IN := #B塔工作A塔待再生_Interval_1);
   END_IF;
   #IEC_Timer_0_Instance7(IN := #CTR_Current_State = 8, PT := #B塔工作A塔待再生_Interval);   // TON
   IF #IEC_Timer_0_Instance7.Q THEN #Cyclic_Switch_Flag := TRUE; END_IF;
END_REGION

REGION Network 20: B塔吸附,A塔热再生(主加热根据温度判断开断;)
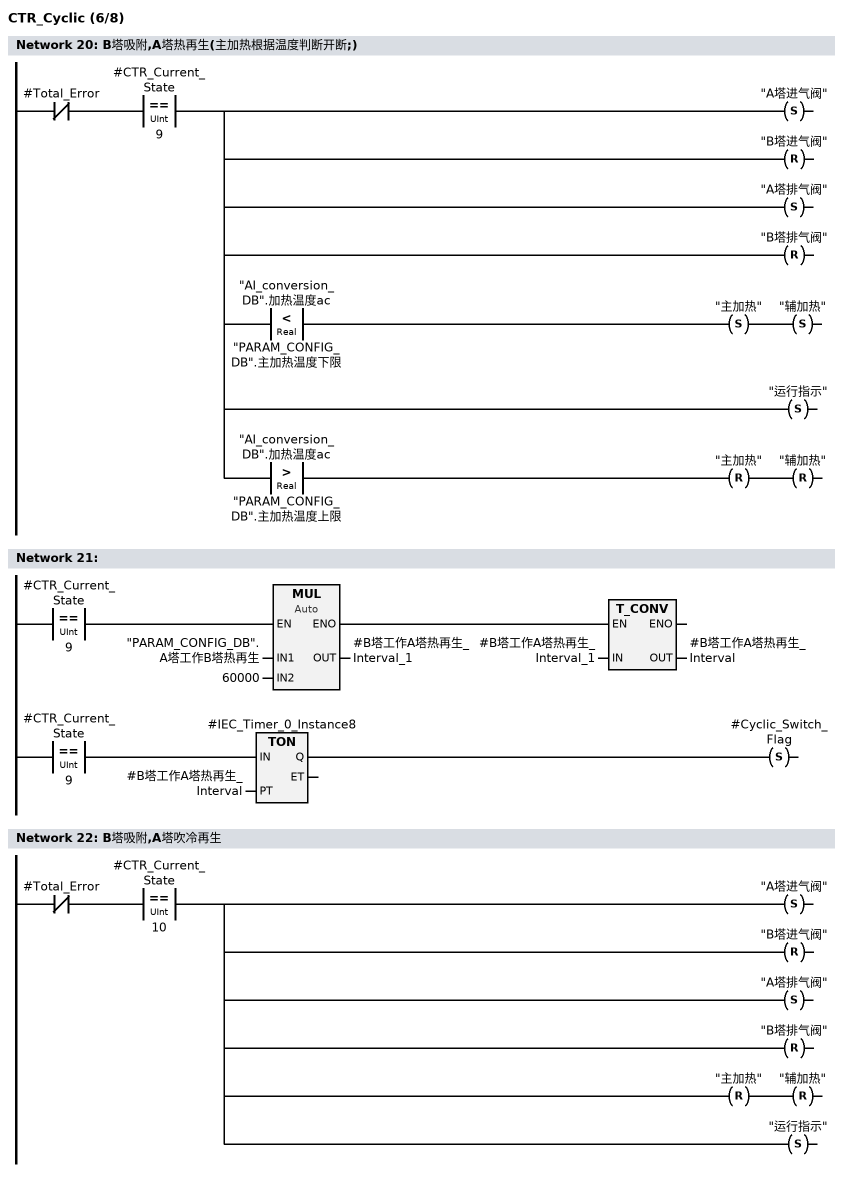
   RUNG wire#powerrail
      I_Contact( #Total_Error )
      { S7_Templates := "SrcType := UInt" } EQ_Contact(in1 := #CTR_Current_State, in2 := 9)
      wire#w1
      S_Coil( "A塔进气阀" )
   END_RUNG
   RUNG wire#w1
      R_Coil( "B塔进气阀" )
   END_RUNG
   RUNG wire#w1
      S_Coil( "A塔排气阀" )
   END_RUNG
   RUNG wire#w1
      R_Coil( "B塔排气阀" )
   END_RUNG
   RUNG wire#w1
      { S7_Templates := "SrcType := Real" } LT_Contact(in1 := "AI_conversion_DB".加热温度ac, in2 := "PARAM_CONFIG_DB".主加热温度下限)
      S_Coil( "主加热" )
      S_Coil( "辅加热" )
   END_RUNG
   RUNG wire#w1
      S_Coil( "运行指示" )
   END_RUNG
   RUNG wire#w1
      { S7_Templates := "SrcType := Real" } GT_Contact(in1 := "AI_conversion_DB".加热温度ac, in2 := "PARAM_CONFIG_DB".主加热温度上限)
      R_Coil( "主加热" )
      R_Coil( "辅加热" )
   END_RUNG
   // the same network as SCL:
   #_w1 := NOT #Total_Error AND (#CTR_Current_State = 9);
   IF #_w1 THEN
       "A塔进气阀" := TRUE;
       "B塔进气阀" := FALSE;
       "A塔排气阀" := TRUE;
       "B塔排气阀" := FALSE;
   END_IF;
   IF #_w1 AND ("AI_conversion_DB".加热温度ac < "PARAM_CONFIG_DB".主加热温度下限) THEN
       "主加热" := TRUE;
       "辅加热" := TRUE;
   END_IF;
   IF #_w1 THEN "运行指示" := TRUE; END_IF;
   IF #_w1 AND ("AI_conversion_DB".加热温度ac > "PARAM_CONFIG_DB".主加热温度上限) THEN
       "主加热" := FALSE;
       "辅加热" := FALSE;
   END_IF;
END_REGION

REGION Network 21
   IF #CTR_Current_State = 9 THEN
       #B塔工作A塔热再生_Interval_1 := "PARAM_CONFIG_DB".A塔工作B塔热再生 * 60000;
       #B塔工作A塔热再生_Interval := T_CONV(IN := #B塔工作A塔热再生_Interval_1);
   END_IF;
   #IEC_Timer_0_Instance8(IN := #CTR_Current_State = 9, PT := #B塔工作A塔热再生_Interval);   // TON
   IF #IEC_Timer_0_Instance8.Q THEN #Cyclic_Switch_Flag := TRUE; END_IF;
END_REGION

REGION Network 22: B塔吸附,A塔吹冷再生
   RUNG wire#powerrail
      I_Contact( #Total_Error )
      { S7_Templates := "SrcType := UInt" } EQ_Contact(in1 := #CTR_Current_State, in2 := 10)
      wire#w1
      S_Coil( "A塔进气阀" )
   END_RUNG
   RUNG wire#w1
      R_Coil( "B塔进气阀" )
   END_RUNG
   RUNG wire#w1
      S_Coil( "A塔排气阀" )
   END_RUNG
   RUNG wire#w1
      R_Coil( "B塔排气阀" )
   END_RUNG
   RUNG wire#w1
      R_Coil( "主加热" )
      R_Coil( "辅加热" )
   END_RUNG
   RUNG wire#w1
      S_Coil( "运行指示" )
   END_RUNG
   // the same network as SCL:
   IF NOT #Total_Error AND (#CTR_Current_State = 10) THEN
       "A塔进气阀" := TRUE;
       "B塔进气阀" := FALSE;
       "A塔排气阀" := TRUE;
       "B塔排气阀" := FALSE;
       "主加热" := FALSE;
       "辅加热" := FALSE;
       "运行指示" := TRUE;
   END_IF;
END_REGION

REGION Network 23
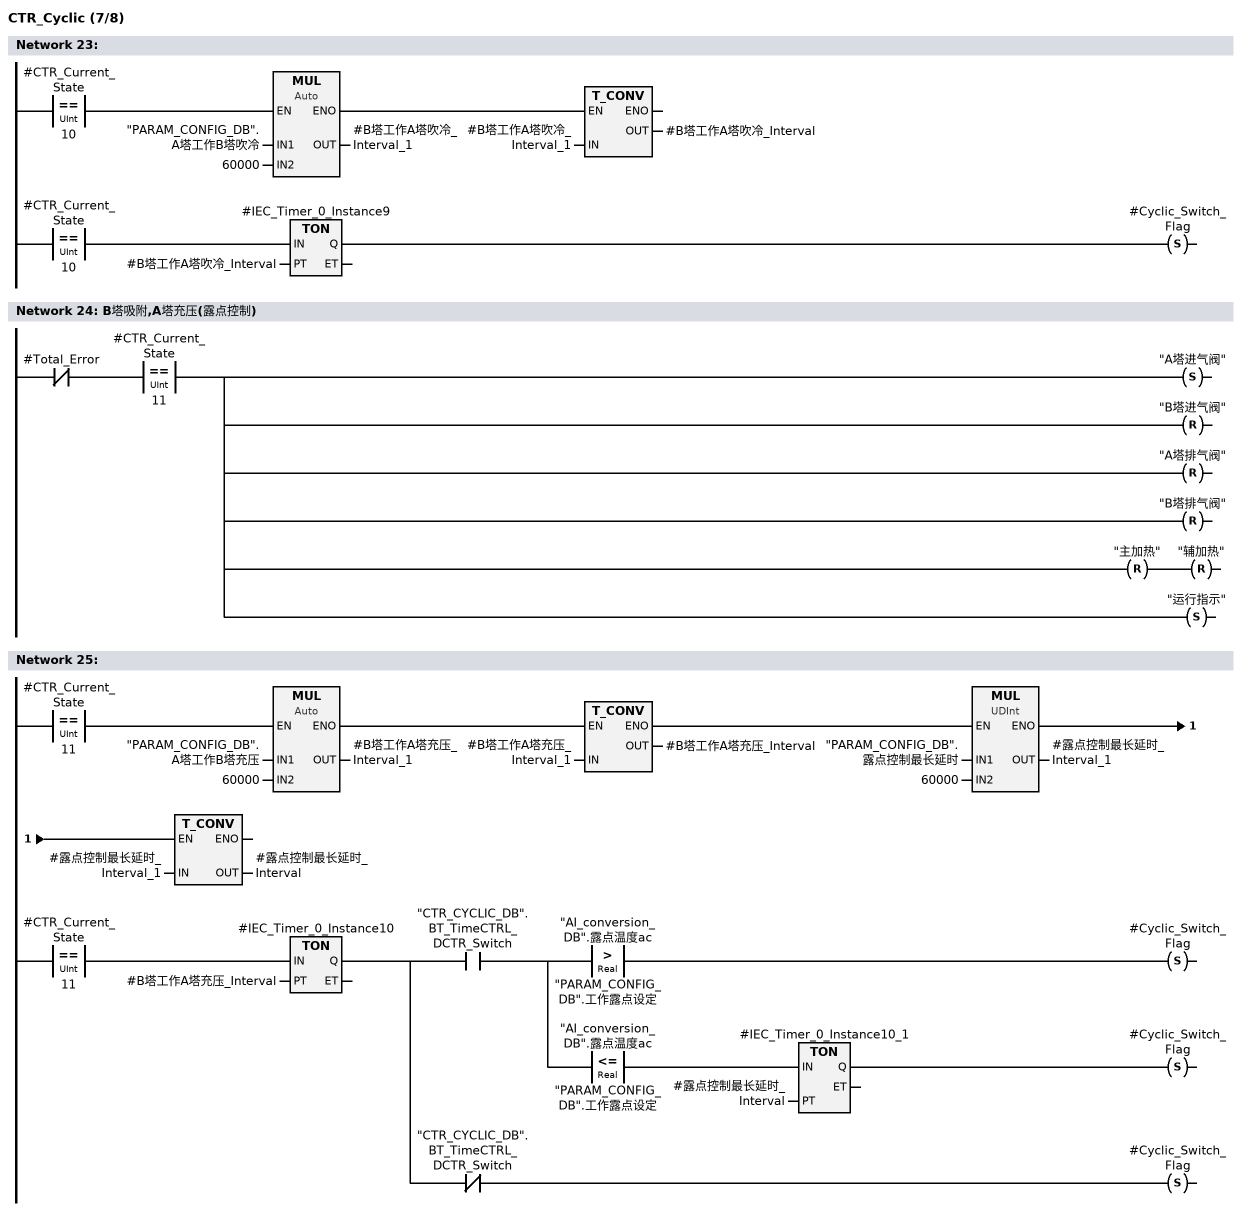
   IF #CTR_Current_State = 10 THEN
       #B塔工作A塔吹冷_Interval_1 := "PARAM_CONFIG_DB".A塔工作B塔吹冷 * 60000;
       #B塔工作A塔吹冷_Interval := T_CONV(IN := #B塔工作A塔吹冷_Interval_1);
   END_IF;
   #IEC_Timer_0_Instance9(IN := #CTR_Current_State = 10, PT := #B塔工作A塔吹冷_Interval);   // TON
   IF #IEC_Timer_0_Instance9.Q THEN #Cyclic_Switch_Flag := TRUE; END_IF;
END_REGION

REGION Network 24: B塔吸附,A塔充压(露点控制)
   RUNG wire#powerrail
      I_Contact( #Total_Error )
      { S7_Templates := "SrcType := UInt" } EQ_Contact(in1 := #CTR_Current_State, in2 := 11)
      wire#w1
      S_Coil( "A塔进气阀" )
   END_RUNG
   RUNG wire#w1
      R_Coil( "B塔进气阀" )
   END_RUNG
   RUNG wire#w1
      R_Coil( "A塔排气阀" )
   END_RUNG
   RUNG wire#w1
      R_Coil( "B塔排气阀" )
   END_RUNG
   RUNG wire#w1
      R_Coil( "主加热" )
      R_Coil( "辅加热" )
   END_RUNG
   RUNG wire#w1
      S_Coil( "运行指示" )
   END_RUNG
   // the same network as SCL:
   IF NOT #Total_Error AND (#CTR_Current_State = 11) THEN
       "A塔进气阀" := TRUE;
       "B塔进气阀" := FALSE;
       "A塔排气阀" := FALSE;
       "B塔排气阀" := FALSE;
       "主加热" := FALSE;
       "辅加热" := FALSE;
       "运行指示" := TRUE;
   END_IF;
END_REGION

REGION Network 25
   // ENO of a box is taken as its EN; it also drops when the box reports an error
   IF #CTR_Current_State = 11 THEN
       #B塔工作A塔充压_Interval_1 := "PARAM_CONFIG_DB".A塔工作B塔充压 * 60000;
       #B塔工作A塔充压_Interval := T_CONV(IN := #B塔工作A塔充压_Interval_1);
       #露点控制最长延时_Interval_1 := "PARAM_CONFIG_DB".露点控制最长延时 * 60000;
       #露点控制最长延时_Interval := T_CONV(IN := #露点控制最长延时_Interval_1);
   END_IF;
   #IEC_Timer_0_Instance10(IN := #CTR_Current_State = 11, PT := #B塔工作A塔充压_Interval);   // TON
   #_w1 := #IEC_Timer_0_Instance10.Q AND "CTR_CYCLIC_DB".BT_TimeCTRL_DCTR_Switch;
   IF #_w1 AND ("AI_conversion_DB".露点温度ac > "PARAM_CONFIG_DB".工作露点设定) THEN
       #Cyclic_Switch_Flag := TRUE;
   END_IF;
   #IEC_Timer_0_Instance10_1(IN := #_w1 AND ("AI_conversion_DB".露点温度ac <= "PARAM_CONFIG_DB".工作露点设定),   // TON
                           PT := #露点控制最长延时_Interval);
   IF #IEC_Timer_0_Instance10_1.Q THEN #Cyclic_Switch_Flag := TRUE; END_IF;
   IF #IEC_Timer_0_Instance10.Q AND NOT "CTR_CYCLIC_DB".BT_TimeCTRL_DCTR_Switch THEN
       #Cyclic_Switch_Flag := TRUE;
   END_IF;
END_REGION

REGION Network 26: B塔吸附,A塔均压
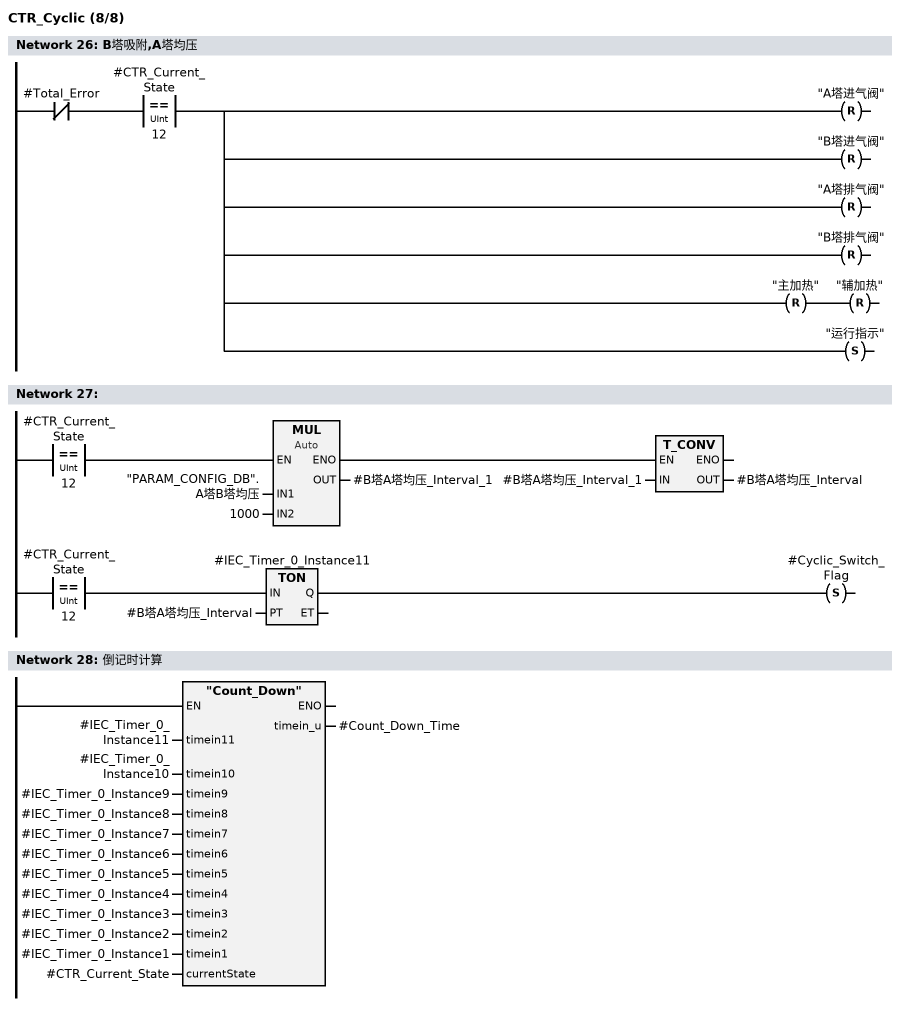
   RUNG wire#powerrail
      I_Contact( #Total_Error )
      { S7_Templates := "SrcType := UInt" } EQ_Contact(in1 := #CTR_Current_State, in2 := 12)
      wire#w1
      R_Coil( "A塔进气阀" )
   END_RUNG
   RUNG wire#w1
      R_Coil( "B塔进气阀" )
   END_RUNG
   RUNG wire#w1
      R_Coil( "A塔排气阀" )
   END_RUNG
   RUNG wire#w1
      R_Coil( "B塔排气阀" )
   END_RUNG
   RUNG wire#w1
      R_Coil( "主加热" )
      R_Coil( "辅加热" )
   END_RUNG
   RUNG wire#w1
      S_Coil( "运行指示" )
   END_RUNG
   // the same network as SCL:
   IF NOT #Total_Error AND (#CTR_Current_State = 12) THEN
       "A塔进气阀" := FALSE;
       "B塔进气阀" := FALSE;
       "A塔排气阀" := FALSE;
       "B塔排气阀" := FALSE;
       "主加热" := FALSE;
       "辅加热" := FALSE;
       "运行指示" := TRUE;
   END_IF;
END_REGION

REGION Network 27
   IF #CTR_Current_State = 12 THEN
       #B塔A塔均压_Interval_1 := "PARAM_CONFIG_DB".A塔B塔均压 * 1000;
       #B塔A塔均压_Interval := T_CONV(IN := #B塔A塔均压_Interval_1);
   END_IF;
   #IEC_Timer_0_Instance11(IN := #CTR_Current_State = 12, PT := #B塔A塔均压_Interval);   // TON
   IF #IEC_Timer_0_Instance11.Q THEN #Cyclic_Switch_Flag := TRUE; END_IF;
END_REGION

REGION Network 28: 倒记时计算
   RUNG wire#powerrail
      "Count_Down"(timein11 := #IEC_Timer_0_Instance11, timein10 := #IEC_Timer_0_Instance10, timein9 := #IEC_Timer_0_Instance9, timein8 := #IEC_Timer_0_Instance8, timein7 := #IEC_Timer_0_Instance7, timein6 := #IEC_Timer_0_Instance6, timein5 := #IEC_Timer_0_Instance5, timein4 := #IEC_Timer_0_Instance4, timein3 := #IEC_Timer_0_Instance3, timein2 := #IEC_Timer_0_Instance2, timein1 := #IEC_Timer_0_Instance1, currentState := #CTR_Current_State, timein_u => #Count_Down_Time)
   END_RUNG
   // the same network as SCL:
   "Count_Down"(timein11 := #IEC_Timer_0_Instance11,
                timein10 := #IEC_Timer_0_Instance10,
                timein9 := #IEC_Timer_0_Instance9,
                timein8 := #IEC_Timer_0_Instance8,
                timein7 := #IEC_Timer_0_Instance7,
                timein6 := #IEC_Timer_0_Instance6,
                timein5 := #IEC_Timer_0_Instance5,
                timein4 := #IEC_Timer_0_Instance4,
                timein3 := #IEC_Timer_0_Instance3,
                timein2 := #IEC_Timer_0_Instance2,
                timein1 := #IEC_Timer_0_Instance1,
                currentState := #CTR_Current_State,
                timein_u => #Count_Down_Time);
END_REGION
END_FUNCTION_BLOCK

FUNCTION_BLOCK "Alarm_Error"   // FB5, LAD
{ S7_Optimized_Access := 'TRUE' }
VERSION : 0.1
   VAR
      AlarmError : UInt;   // 0:进气气压报警位;
      PRE_AlarmErrorX5 : Bool;
      PRE_AlarmErrorX4 : Bool;
      PRE_AlarmErrorX3 : Bool;
      PRE_AlarmErrorX2 : Bool;
      PRE_AlarmErrorX1 : Bool;
      PRE_AlarmErrorX0 : Bool;
      IEC_Timer_0_Instance : TON_TIME;
      IEC_Timer_0_Instance_1 : TON_TIME;
      IEC_Timer_0_Instance_2 : TON_TIME;
      IEC_Timer_0_Instance_3 : TON_TIME;
      IEC_Timer_0_Instance_4 : TON_TIME;
   END_VAR
   VAR_TEMP
      ErrorDelayInterval_ud : UDInt;
      ErrorDelayInterval_t : Time;
   END_VAR
   VAR_TEMP   // added for the SCL form of the ladder/FBD networks
      _w1 : Bool;
      _w2 : Bool;
      _w3 : Bool;
   END_VAR
BEGIN

REGION Network 1: 故障延时判断
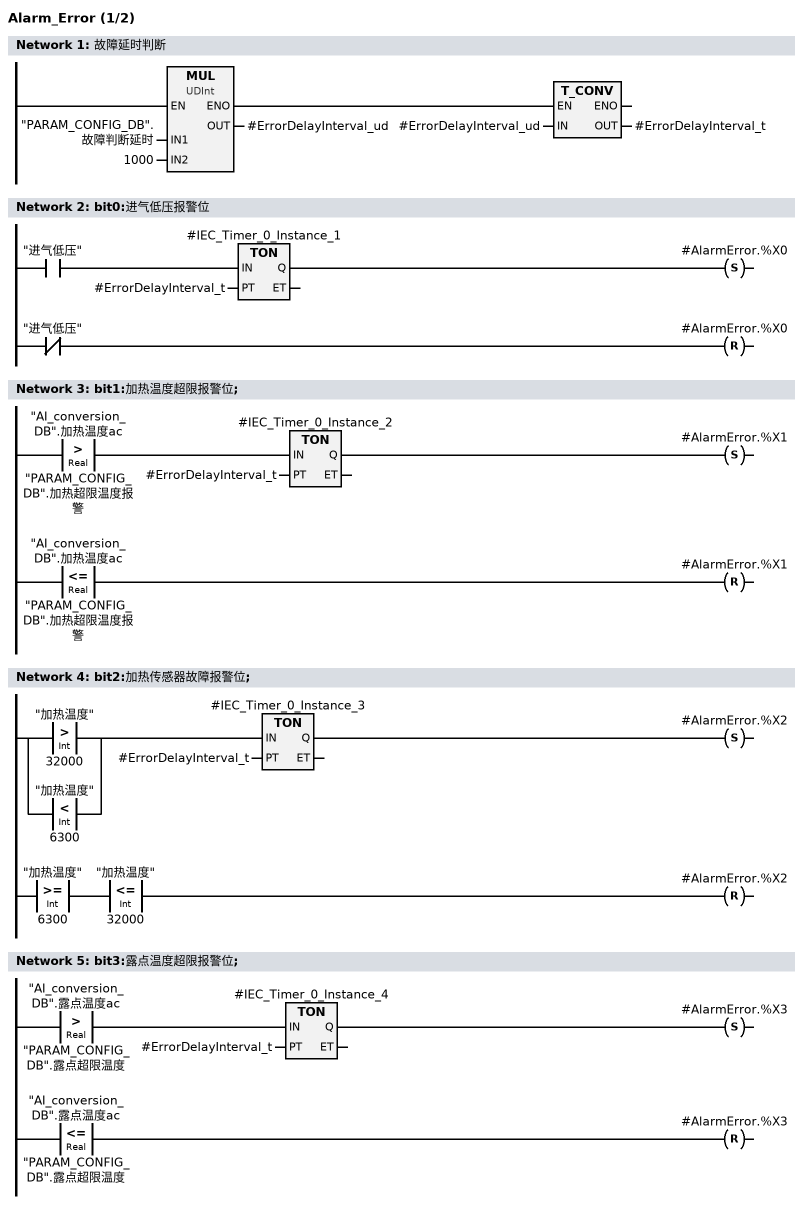
   #ErrorDelayInterval_ud := "PARAM_CONFIG_DB".故障判断延时 * 1000;
   #ErrorDelayInterval_t := T_CONV(IN := #ErrorDelayInterval_ud);
END_REGION

REGION Network 2: bit0:进气低压报警位
   #IEC_Timer_0_Instance_1(IN := "进气低压", PT := #ErrorDelayInterval_t);   // TON
   IF #IEC_Timer_0_Instance_1.Q THEN #AlarmError.%X0 := TRUE; END_IF;
   IF NOT "进气低压" THEN #AlarmError.%X0 := FALSE; END_IF;
END_REGION

REGION Network 3: bit1:加热温度超限报警位;
   #IEC_Timer_0_Instance_2(IN := "AI_conversion_DB".加热温度ac > "PARAM_CONFIG_DB".加热超限温度报警,   // TON
                           PT := #ErrorDelayInterval_t);
   IF #IEC_Timer_0_Instance_2.Q THEN #AlarmError.%X1 := TRUE; END_IF;
   IF "AI_conversion_DB".加热温度ac <= "PARAM_CONFIG_DB".加热超限温度报警 THEN #AlarmError.%X1 := FALSE; END_IF;
END_REGION

REGION Network 4: bit2:加热传感器故障报警位;
   #IEC_Timer_0_Instance_3(IN := ("加热温度" > 32000) OR ("加热温度" < 6300), PT := #ErrorDelayInterval_t);   // TON
   IF #IEC_Timer_0_Instance_3.Q THEN #AlarmError.%X2 := TRUE; END_IF;
   IF ("加热温度" >= 6300) AND ("加热温度" <= 32000) THEN #AlarmError.%X2 := FALSE; END_IF;
END_REGION

REGION Network 5: bit3:露点温度超限报警位;
   #IEC_Timer_0_Instance_4(IN := "AI_conversion_DB".露点温度ac > "PARAM_CONFIG_DB".露点超限温度,   // TON
                           PT := #ErrorDelayInterval_t);
   IF #IEC_Timer_0_Instance_4.Q THEN #AlarmError.%X3 := TRUE; END_IF;
   IF "AI_conversion_DB".露点温度ac <= "PARAM_CONFIG_DB".露点超限温度 THEN #AlarmError.%X3 := FALSE; END_IF;
END_REGION

REGION Network 6: 报警停机操作
   // 露点报警不做停机操作
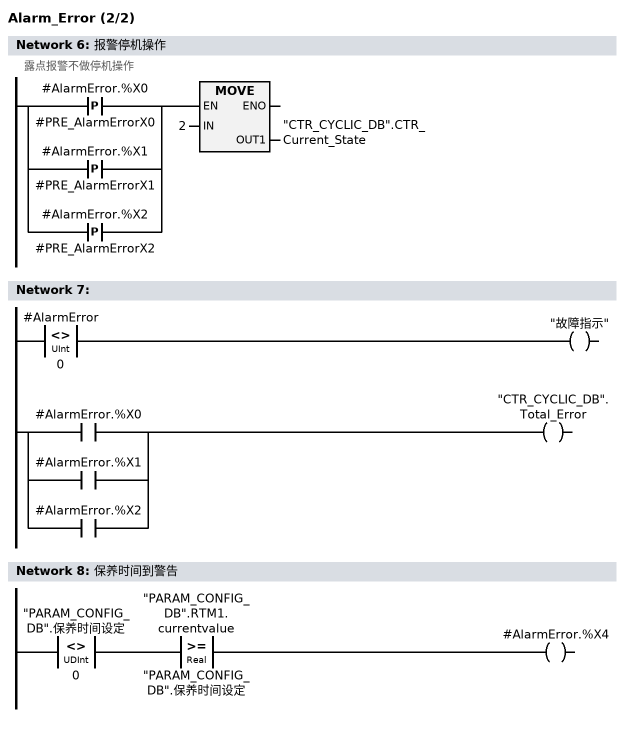
   RUNG wire#powerrail
      P_Contact(operand := #AlarmError.%X0, bit := #PRE_AlarmErrorX0)
      wire#w1
      Move(in := 2, out1 => "CTR_CYCLIC_DB".CTR_Current_State)
   END_RUNG
   RUNG wire#powerrail
      P_Contact(operand := #AlarmError.%X1, bit := #PRE_AlarmErrorX1)
   END_RUNG wire#w1
   RUNG wire#powerrail
      P_Contact(operand := #AlarmError.%X2, bit := #PRE_AlarmErrorX2)
   END_RUNG wire#w1
   // the same network as SCL:
   #_w1 := #AlarmError.%X0 AND NOT #PRE_AlarmErrorX0;   // rising edge of #AlarmError.%X0
   #PRE_AlarmErrorX0 := #AlarmError.%X0;
   #_w2 := #AlarmError.%X1 AND NOT #PRE_AlarmErrorX1;   // rising edge of #AlarmError.%X1
   #PRE_AlarmErrorX1 := #AlarmError.%X1;
   #_w3 := #AlarmError.%X2 AND NOT #PRE_AlarmErrorX2;   // rising edge of #AlarmError.%X2
   #PRE_AlarmErrorX2 := #AlarmError.%X2;
   IF #_w1 OR #_w2 OR #_w3 THEN "CTR_CYCLIC_DB".CTR_Current_State := 2; END_IF;
END_REGION

REGION Network 7
   RUNG wire#powerrail
      { S7_Templates := "SrcType := UInt" } NE_Contact(in1 := #AlarmError, in2 := 0)
      Coil( "故障指示" )
   END_RUNG
   RUNG wire#powerrail
      Contact( #AlarmError.%X0 )
      wire#w1
      Coil( "CTR_CYCLIC_DB".Total_Error )
   END_RUNG
   RUNG wire#powerrail
      Contact( #AlarmError.%X1 )
   END_RUNG wire#w1
   RUNG wire#powerrail
      Contact( #AlarmError.%X2 )
   END_RUNG wire#w1
   // the same network as SCL:
   "故障指示" := #AlarmError <> 0;
   "CTR_CYCLIC_DB".Total_Error := #AlarmError.%X0 OR #AlarmError.%X1 OR #AlarmError.%X2;
END_REGION

REGION Network 8: 保养时间到警告
   RUNG wire#powerrail
      { S7_Templates := "SrcType := UDInt" } NE_Contact(in1 := "PARAM_CONFIG_DB".保养时间设定, in2 := 0)
      { S7_Templates := "SrcType := Real" } GE_Contact(in1 := "PARAM_CONFIG_DB".RTM1.currentvalue, in2 := "PARAM_CONFIG_DB".保养时间设定)
      Coil( #AlarmError.%X4 )
   END_RUNG
   // the same network as SCL:
   #AlarmError.%X4 := ("PARAM_CONFIG_DB".保养时间设定 <> 0) AND ("PARAM_CONFIG_DB".RTM1.currentvalue >= "PARAM_CONFIG_DB".保养时间设定);
END_REGION
END_FUNCTION_BLOCK

FUNCTION "Cyclic_Switch" : Void   // FC1, SCL
{ S7_Optimized_Access := 'TRUE' }
VERSION : 0.1
   VAR_INPUT
      Cyclic_Switch_Enable : Bool;
      Current_State : UInt;
   END_VAR
   VAR_OUTPUT
      Cyclic_Switch_Reset : Bool;
      Current_State_Output : UInt;
   END_VAR
BEGIN
   IF #Cyclic_Switch_Enable = TRUE THEN
       IF #Current_State = 2 THEN
           #Current_State := 0;

       ELSIF #Current_State >= 3 THEN
           IF #Current_State < 12 THEN
               #Current_State := #Current_State + 1;
           ELSE
               #Current_State := 3;
           END_IF;
       END_IF;
       #Cyclic_Switch_Reset := FALSE;
       //#Current_State_Output := #Current_State;
   END_IF;
   #Current_State_Output := #Current_State;
END_FUNCTION

FUNCTION "Count_Down" : Void   // FC2, SCL
{ S7_Optimized_Access := 'TRUE' }
VERSION : 0.1
   VAR_INPUT
      timein11 : IEC_TIMER;
      timein10 : IEC_TIMER;
      timein9 : IEC_TIMER;
      timein8 : IEC_TIMER;
      timein7 : IEC_TIMER;
      timein6 : IEC_TIMER;
      timein5 : IEC_TIMER;
      timein4 : IEC_TIMER;
      timein3 : IEC_TIMER;
      timein2 : IEC_TIMER;
      timein1 : IEC_TIMER;
      currentState : UInt;
   END_VAR
   VAR_OUTPUT
      timein_u : UDInt;   // s
   END_VAR
   VAR_TEMP
      timein_t : Time;
   END_VAR
BEGIN
   IF #currentState = 2 THEN
       #timein_t := #timein1.PT - #timein1.ET;
   ELSIF #currentState = 3 THEN
       #timein_t := #timein2.PT - #timein2.ET;
   ELSIF #currentState = 4 THEN
       #timein_t := #timein3.PT - #timein3.ET;
   ELSIF #currentState = 5 THEN
       #timein_t := #timein4.PT - #timein4.ET;
   ELSIF #currentState = 6 THEN
       #timein_t := #timein5.PT - #timein5.ET;
   ELSIF #currentState = 7 THEN
       #timein_t := #timein6.PT - #timein5.ET;
   ELSIF #currentState = 8 THEN
       #timein_t := #timein7.PT - #timein7.ET;
   ELSIF #currentState = 9 THEN
       #timein_t := #timein8.PT - #timein8.ET;
   ELSIF #currentState = 10 THEN
       #timein_t := #timein9.PT - #timein9.ET;
   ELSIF #currentState = 11 THEN
       #timein_t := #timein10.PT - #timein10.ET;
   ELSIF #currentState = 12 THEN
       #timein_t := #timein11.PT - #timein11.ET;
   ELSE
       #timein_t := T#0ms;
   END_IF;
   #timein_u := T_CONV(#timein_t)/1000;//s
END_FUNCTION

// folder: ModbusRTU

FUNCTION_BLOCK "modbusrtu"   // FB1, LAD
{ S7_Optimized_Access := 'TRUE' }
VERSION : 0.1
   VAR
      MB_SLAVE_STATUS : Struct
         NDR : Bool;
         DR : Bool;
         PRE_ERROR : Bool;
         ERROR : Bool;
         STATUS : UInt;
      END_STRUCT;
   END_VAR
   VAR_TEMP   // added for the SCL form of the ladder/FBD networks
      _w1 : Bool;
   END_VAR
BEGIN

REGION Network 1
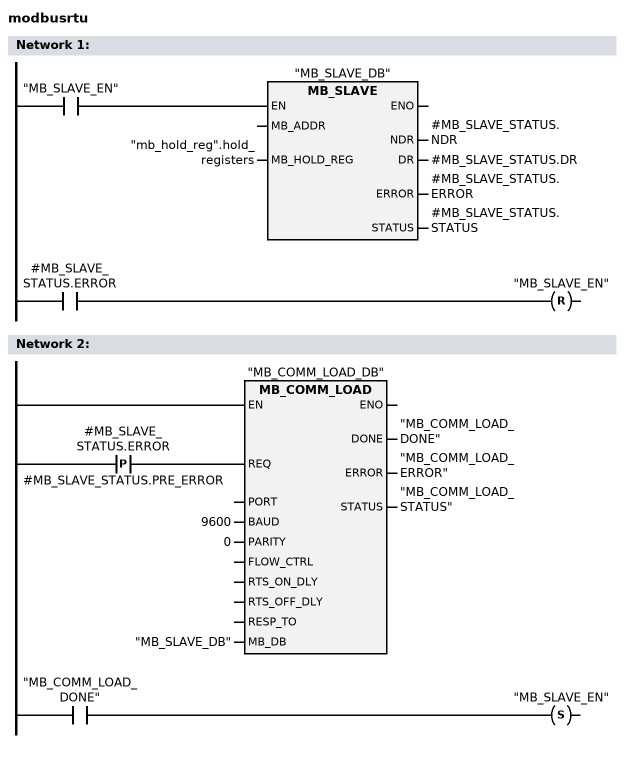
   IF "MB_SLAVE_EN" THEN
       "MB_SLAVE_DB"(MB_HOLD_REG := "mb_hold_reg".hold_registers,   // MB_SLAVE
                     NDR => #MB_SLAVE_STATUS.NDR,
                     DR => #MB_SLAVE_STATUS.DR,
                     ERROR => #MB_SLAVE_STATUS.ERROR,
                     STATUS => #MB_SLAVE_STATUS.STATUS);
   END_IF;
   IF #MB_SLAVE_STATUS.ERROR THEN "MB_SLAVE_EN" := FALSE; END_IF;
END_REGION

REGION Network 2
   #_w1 := #MB_SLAVE_STATUS.ERROR AND NOT #MB_SLAVE_STATUS.PRE_ERROR;   // rising edge of #MB_SLAVE_STATUS.ERROR
   #MB_SLAVE_STATUS.PRE_ERROR := #MB_SLAVE_STATUS.ERROR;
   "MB_COMM_LOAD_DB"(REQ := #_w1,   // MB_COMM_LOAD
                     BAUD := 9600,
                     PARITY := 0,
                     MB_DB := "MB_SLAVE_DB",
                     DONE => "MB_COMM_LOAD_DONE",
                     ERROR => "MB_COMM_LOAD_ERROR",
                     STATUS => "MB_COMM_LOAD_STATUS");
   IF "MB_COMM_LOAD_DONE" THEN "MB_SLAVE_EN" := TRUE; END_IF;
END_REGION
END_FUNCTION_BLOCK

(* ===== HMI "HMI_RT_2" =====
system functions are stored by id; their names below are inferred from use
connection "HMI_连接_2": ETHERNET, SMART_S7_1200_OMS

HMI tags "默认变量表"
   "Tag_ScreenNumber" : UInt, internal
   "加热温度" : Int = PLC 加热温度 AT %IW66, 1 s
   "AlarmError_DB_AlarmError" : UInt = PLC AlarmError_DB.AlarmError, 1 s
   "PARAM_CONFIG_DB_BT_Function_BT_Runtime_Reset" : Bool = PLC PARAM_CONFIG_DB.BT_Function.BT_Runtime_Reset AT %DB1.DBX0.0, 1 s
   "CTR_CYCLIC_DB_BT_function_BT_Atower_Open" : Bool = PLC CTR_CYCLIC_DB.BT_function.BT_Atower_Open AT %DB1.DBX0.0, 1 s
   "CTR_CYCLIC_DB_BT_function_BT_Btower_Open" : Bool = PLC CTR_CYCLIC_DB.BT_function.BT_Btower_Open AT %DB1.DBX0.0, 1 s
   "CTR_CYCLIC_DB_BT_function_BT_Stop" : Bool = PLC CTR_CYCLIC_DB.BT_function.BT_Stop AT %DB1.DBX0.0, 1 s
   "CTR_CYCLIC_DB_CTR_Current_State" : UInt = PLC CTR_CYCLIC_DB.CTR_Current_State, 1 s
   "CTR_CYCLIC_DB_Count_Down_Time" : UDInt = PLC CTR_CYCLIC_DB.Count_Down_Time, 1 s
   "CTR_CYCLIC_DB_BT_LocalRemoteSwitch" : Bool = PLC CTR_CYCLIC_DB.BT_LocalRemoteSwitch AT %DB1.DBW0, 1 s
   "CTR_CYCLIC_DB_BT_TimeCTRL_DCTR_Switch" : Bool = PLC CTR_CYCLIC_DB.BT_TimeCTRL_DCTR_Switch AT %DB1.DBX0.0, 1 s
   "PARAM_CONFIG_DB_MaintainTime_CountdownValue" : Real = PLC PARAM_CONFIG_DB.MaintainTime_CountdownValue AT %DB1.DBW0, 1 s

HMI tags "PLC_Variables"
   "A塔进气阀" : Bool = PLC A塔进气阀 AT %Q0.0, 1 s
   "A塔排气阀" : Bool = PLC A塔排气阀 AT %Q0.2, 1 s
   "B塔进气阀" : Bool = PLC B塔进气阀 AT %Q0.1, 1 s
   "B塔排气阀" : Bool = PLC B塔排气阀 AT %Q0.3, 1 s
   "本地远程转换" : Bool = PLC 本地远程转换 AT %I0.2, 1 s
   "辅加热" : Bool = PLC 辅加热 AT %Q0.5, 1 s
   "故障指示" : Bool = PLC 故障指示 AT %Q0.7, 1 s
   "进气低压" : Bool = PLC 进气低压 AT %I0.6, 1 s
   "开机" : Bool = PLC 开机 AT %I0.0, 1 s
   "停机" : Bool = PLC 停机 AT %I0.1, 1 s
   "远程开机" : Bool = PLC 远程开机 AT %I0.3, 1 s
   "远程停机" : Bool = PLC 远程停机 AT %I0.4, 1 s
   "远程指示" : Bool = PLC 远程指示 AT %Q1.0, 1 s
   "运行指示" : Bool = PLC 运行指示 AT %Q0.6, 1 s
   "主加热" : Bool = PLC 主加热 AT %Q0.4, 1 s
   "AI_conversion_DB_露点温度ac" : Real = PLC AI_conversion_DB.露点温度ac, 1 s
   "AI_conversion_DB_加热温度ac" : Real = PLC AI_conversion_DB.加热温度ac, 1 s
   "PARAM_CONFIG_DB_主加热温度上限" : UInt = PLC PARAM_CONFIG_DB.主加热温度上限 AT %DB1.DBX0.0, 1 s
   "PARAM_CONFIG_DB_主加热温度下限" : UInt = PLC PARAM_CONFIG_DB.主加热温度下限 AT %DB1.DBW0, 1 s
   "PARAM_CONFIG_DB_加热超限温度报警" : UInt = PLC PARAM_CONFIG_DB.加热超限温度报警 AT %DB1.DBW0, 1 s
   "PARAM_CONFIG_DB_露点超限温度" : Int = PLC PARAM_CONFIG_DB.露点超限温度 AT %DB1.DBW0, 1 s
   "PARAM_CONFIG_DB_加热温度补偿" : Int = PLC PARAM_CONFIG_DB.加热温度补偿 AT %DB1.DBW0, 1 s
   "PARAM_CONFIG_DB_压力温度补偿" : Int = PLC PARAM_CONFIG_DB.压力温度补偿 AT %DB1.DBW0, 1 s
   "PARAM_CONFIG_DB_工作露点设定" : Int = PLC PARAM_CONFIG_DB.工作露点设定 AT %DB1.DBW0, 1 s
   "PARAM_CONFIG_DB_停机充压时间" : UDInt = PLC PARAM_CONFIG_DB.停机充压时间 AT %DB1.DBW0, 1 s
   "PARAM_CONFIG_DB_A塔工作B塔待再生" : UDInt = PLC PARAM_CONFIG_DB.A塔工作B塔待再生 AT %DB1.DBW0, 1 s
   "PARAM_CONFIG_DB_A塔工作B塔热再生" : UDInt = PLC PARAM_CONFIG_DB.A塔工作B塔热再生 AT %DB1.DBW0, 1 s
   "PARAM_CONFIG_DB_A塔工作B塔吹冷" : UDInt = PLC PARAM_CONFIG_DB.A塔工作B塔吹冷 AT %DB1.DBW0, 1 s
   "PARAM_CONFIG_DB_A塔工作B塔充压" : UDInt = PLC PARAM_CONFIG_DB.A塔工作B塔充压 AT %DB1.DBW0, 1 s
   "PARAM_CONFIG_DB_A塔B塔均压" : UDInt = PLC PARAM_CONFIG_DB.A塔B塔均压 AT %DB1.DBW0, 1 s
   "PARAM_CONFIG_DB_故障判断延时" : UInt = PLC PARAM_CONFIG_DB.故障判断延时 AT %DB1.DBW0, 1 s
   "PARAM_CONFIG_DB_保养时间设定" : UDInt = PLC PARAM_CONFIG_DB.保养时间设定 AT %DB1.DBW0, 1 s
   "PARAM_CONFIG_DB_从站地址" : UInt = PLC PARAM_CONFIG_DB.从站地址 AT %DB1.DBD0, 1 s
   "PARAM_CONFIG_DB_露点控制最长延时" : UInt = PLC PARAM_CONFIG_DB.露点控制最长延时 AT %DB1.DBW0, 1 s
   "PARAM_CONFIG_DB_RTM1_currentvalue" : DInt = PLC PARAM_CONFIG_DB.RTM1.currentvalue AT %DB1.DBW0, 1 s

discrete alarms
   1: '进气低压报警', class Errors, trigger "AlarmError_DB_AlarmError" bit 0
   2: '系统运行时间超过保养时间!', class Warnings, trigger "AlarmError_DB_AlarmError" bit 4

analog alarms
   1: '加热温度超过限制报警值', class Errors, trigger "AI_conversion_DB_加热温度ac"
   2: '加热传感器故障', class Errors, trigger "加热温度"
   3: '加热传感器故障', class Errors, trigger "加热温度"
   4: '露点温度超过限制报警值', class Warnings, trigger "AI_conversion_DB_露点温度ac"

text list "远程就地": 0 '就地'; 1 '远程'

text list "露点时间控制": 1 '露点控制'; 0 '时间控制'

text list "循环控制状态": 0 '准备就绪'; 2 '停机充压中'; 3 'A塔吸附,B塔待再生'; 4 'A塔吸附,B塔热再生'; 5 'A塔吸附,B塔冷再生'; 6 'A塔吸附,B塔充压'; 7 'A塔吸附,B塔均压'; 8 'B塔吸附,A塔待再生'; 9 'B塔吸附,A塔热再生'; 10 'B塔吸附,A塔冷再生'; 11 'B塔吸附,A塔充压'; 12 'B塔吸附,A塔均压'

graphic list "value1": 0 '图形_26'; 1 '图形_25'

graphic list "value2": 0 '图形_25'; 1 '图形_26'

Template "Template_1" 800x480
   Button "退出" at 714,429 size 71x50; TextOff '退出'; PictureOff "ExitRuntime_KTP700_Basic_PN_TR"; PictureOn "ExitRuntime_KTP700_Basic_PN_TR"; Authorization "Operate"
      on Release: StopRuntime(0)
   Button "登录" at 514,429 size 71x50; TextOff '登录'; PictureOff "Login_KTP700_Basic_PN_TR"; PictureOn "Login_KTP700_Basic_PN_TR"; Authorization "Operate"
      on Release: ActivateScreen("用户管理", 0)
   Button "语言" at 414,429 size 71x50; TextOff 'Text'; PictureOff "ToggleLanguage_KTP700_Basic_PN_TR"; PictureOn "ToggleLanguage_KTP700_Basic_PN_TR"
   Button "Template_Button" at 615,429 size 71x50; TextOff 'Text'; PictureOff "back"
      on Release: function_efd93a16()
   Button "Template_Button_1" at 314,429 size 71x50; TextOff 'Text'; PictureOff "config"; Authorization "Operate"
      on Release: ActivateScreen("参数配置", 0)
   Button "Template_Button_2" at 214,429 size 71x50; TextOff 'Text'; PictureOff "trend"
      on Release: ActivateScreen("趋势", 0)
   Button "报警" at 114,429 size 71x50; TextOff '报警'; PictureOff "AlarmDisplay_KTP700_Basic_PN_TR"; PictureOn "AlarmDisplay_KTP700_Basic_PN_TR"
      on Release: ActivateScreen("报警", 0)
   Button "起始画面" at 14,429 size 71x50; TextOff '起始画面'; PictureOff "NavigateHome_KTP700_Basic_PN_TR"; PictureOn "NavigateHome_KTP700_Basic_PN_TR"
      on Release: ActivateScreen("根画面", 0)
   DateTimeField "HmiScreenItemData" at 691,0 size 105x25
   DateTimeField "HmiScreenItemData_1" at 592,0 size 105x25
   GraphicView "Logo" at 0,0 size 91x51; Picture "HMI_2 的 Logo"
   TextField "文本域_8" at 617,28 size 88x18; Text '系统已运行'
   TextField "文本域_9" at 757,28 size 37x18; Text '小时'
   IOField "I/O 域_4" at 704,27 size 55x22; FormatPattern s99999
      ProcessValue <- "PARAM_CONFIG_DB_RTM1_currentvalue"

screen "根画面" 800x480, template "Template_1"
   on GenerateScreen: SetTag("Tag_ScreenNumber", 1)
   GraphicView "图形视图_11" at 497,172 size 80x128; Picture "图形_3"
   GraphicView "图形视图_3" at 636,269 size 25x55; Picture "图形_7"
   GraphicView "图形视图_4" at 599,185 size 51x73; Picture "图形_8"
   GraphicView "图形视图_5" at 711,172 size 80x128; Picture "图形_3"
   GraphicView "图形视图_14" at 540,104 size 39x22; Picture "图形_11"
   GraphicView "图形视图_15" at 526,105 size 21x20; Picture "图形_13"
   GraphicView "图形视图_16" at 525,120 size 22x55; Picture "图形_14"
   GraphicView "图形视图_17" at 540,147 size 39x21; Picture "图形_11"
   GraphicView "图形视图_18" at 645,146 size 23x23; Picture "图形_15"
   GraphicView "图形视图_19" at 609,147 size 39x21; Picture "图形_11"
   GraphicView "图形视图_20" at 665,147 size 22x21; Picture "图形_11"
   GraphicView "图形视图_21" at 647,226 size 20x20; Picture "图形_16"
   GraphicView "图形视图_22" at 645,166 size 23x65; Picture "图形_14"
   GraphicView "图形视图_23" at 645,103 size 23x23; Picture "图形_17"
   GraphicView "图形视图_24" at 609,104 size 39x21; Picture "图形_11"
   GraphicView "图形视图_25" at 667,104 size 20x21; Picture "图形_11"
   GraphicView "图形视图_26" at 570,238 size 35x20; Picture "图形_11"
   GraphicView "图形视图_27" at 645,73 size 23x33; Picture "图形_14"
   GraphicView "图形视图_28" at 645,53 size 22x22; Picture "图形_18"
   GraphicView "图形视图_29" at 443,54 size 204x21; Picture "图形_11"
   GraphicView "图形视图_9" at 468,67 size 23x178; Picture "图形_14"
   GraphicView "图形视图_30" at 468,237 size 23x23; Picture "图形_19"
   GraphicView "图形视图_31" at 486,238 size 17x20; Picture "图形_11"
   TextField "文本域_4" at 526,225 size 18x27; Text 'A'
   TextField "文本域_5" at 743,223 size 18x27; Text 'B'
   GraphicView "图形视图_32" at 716,147 size 32x21; Picture "图形_11"
   GraphicView "图形视图_33" at 715,104 size 29x21; Picture "图形_11"
   GraphicView "图形视图_34" at 738,104 size 22x22; Picture "图形_18"
   GraphicView "图形视图_35" at 738,123 size 23x52; Picture "图形_14"
   GraphicView "图形视图_36" at 541,335 size 41x21; Picture "图形_11"
   GraphicView "图形视图_37" at 525,296 size 22x85; Picture "图形_14"
   GraphicView "图形视图_38" at 543,378 size 39x20; Picture "图形_11"
   GraphicView "图形视图_39" at 637,377 size 23x22; Picture "图形_15"
   GraphicView "图形视图_40" at 610,378 size 41x20; Picture "图形_11"
   GraphicView "图形视图_41" at 658,378 size 31x20; Picture "图形_11"
   GraphicView "图形视图_42" at 637,334 size 23x22; Picture "图形_17"
   GraphicView "图形视图_43" at 611,335 size 40x20; Picture "图形_11"
   GraphicView "图形视图_44" at 657,335 size 32x20; Picture "图形_11"
   GraphicView "图形视图_45" at 719,378 size 32x20; Picture "图形_11"
   GraphicView "图形视图_46" at 718,335 size 29x20; Picture "图形_11"
   GraphicView "图形视图_49" at 741,296 size 22x85; Picture "图形_14"
   GraphicView "图形视图_50" at 739,376 size 24x24; Picture "图形_16"
   GraphicView "图形视图_51" at 525,377 size 22x22; Picture "图形_19"
   GraphicView "图形视图_52" at 637,324 size 23x13; Picture "图形_14"
   GraphicView "图形视图_53" at 637,397 size 22x22; Picture "图形_16"
   GraphicView "图形视图_54" at 447,399 size 191x20; Picture "图形_11"
   GraphicView "图形视图_48" at 393,383 size 57x57; Picture "图形_21"
   GraphicView "图形视图_47" at 394,38 size 55x55; Picture "图形_20"
   TrendView "趋势视图_1" at 0,185 size 344x172
   Button "Template_Button_2" at 16,366 size 71x50; TextOff 'A塔开机 / A Open'
      on Press: SetBit("CTR_CYCLIC_DB_BT_function_BT_Atower_Open")
      on Release: ResetBit("CTR_CYCLIC_DB_BT_function_BT_Atower_Open")
   Button "Template_Button_1" at 96,366 size 71x50; TextOff 'B塔开机 / B Open'
      on Press: SetBit("CTR_CYCLIC_DB_BT_function_BT_Btower_Open")
      on Release: ResetBit("CTR_CYCLIC_DB_BT_function_BT_Btower_Open")
   Button "Template_Button_3" at 176,366 size 71x50; TextOff '停止 / Stop'
      on Press: SetBit("CTR_CYCLIC_DB_BT_function_BT_Stop")
      on Release: ResetBit("CTR_CYCLIC_DB_BT_function_BT_Stop")
   Button "Template_Button_4" at 256,366 size 71x50; TextOff 'Text'; TextList "远程就地"; Authorization "Operate"
      ProcessValue <- "CTR_CYCLIC_DB_BT_LocalRemoteSwitch"
   TextField "文本域_1" at 46,59 size 263x20; Text '微热吸附式干燥机控制面板'
   TextField "文本域_2" at 34,162 size 63x20; Text '加热器 / Heater'
   TextField "文本域_3" at 146,162 size 190x20; Text '吸附时间与倒计时时间 / Adsorption&Countdown'
   Circle "圆_1" at 52,136 size 23x23
      Appearance <- "主加热"
   IOField "I/O 域_1" at 163,131 size 139x30; FormatPattern 9999999999
      ProcessValue <- "CTR_CYCLIC_DB_Count_Down_Time"
   Group "Group" at 393,38 size 398x402; Picture "图形_3"; Text 'Text'
   TextField "文本域_6" at 376,100 size 104x20; Text '露点温度: / Dew point TEM:'
   IOField "I/O 域_2" at 377,121 size 83x31; FormatPattern s999999999.9
      ProcessValue <- "AI_conversion_DB_露点温度ac"
   TextField "文本域_7" at 377,166 size 70x20; Text '加热温度: / Heat TEM:'
   IOField "I/O 域_3" at 378,186 size 82x31; FormatPattern s999999999.9
      ProcessValue <- "AI_conversion_DB_加热温度ac"
   GraphicView "图形视图_55" at 638,334 size 21x22; Picture "图形_17"
   GraphicView "图形视图_56" at 637,377 size 22x22; Picture "图形_15"
   Button "Template_Button_5" at 377,306 size 93x50; TextOff 'Text'; TextList "露点时间控制"; Authorization "Operate"
      on Click: InvertBit("CTR_CYCLIC_DB_BT_TimeCTRL_DCTR_Switch")
      ProcessValue <- "CTR_CYCLIC_DB_BT_TimeCTRL_DCTR_Switch"
   SymbolicIOField "符号 I/O 域_1" at 16,94 size 311x32; TextOff '0'; TextOn '1'; TextList "循环控制状态"
      ProcessValue <- "CTR_CYCLIC_DB_CTR_Current_State"
   GraphicIOField "图形 I/O 域_1" at 574,368 size 41x34; PictureList "value1"
      ProcessValue <- "A塔进气阀"
   GraphicIOField "图形 I/O 域_2" at 686,369 size 41x34; PictureList "value1"
      ProcessValue <- "B塔进气阀"
   GraphicIOField "图形 I/O 域_3" at 574,325 size 41x34; PictureList "value2"
      ProcessValue <- "A塔排气阀"
   GraphicIOField "图形 I/O 域_4" at 686,326 size 41x34; PictureList "value2"
      ProcessValue <- "B塔排气阀"
   GraphicView "图形视图_1" at 574,84 size 37x43; Picture "图形_29"
   GraphicView "图形视图_2" at 680,83 size 37x43; Picture "图形_29"
   GraphicView "图形视图_6" at 575,128 size 37x43; Picture "图形_29"
   GraphicView "图形视图_7" at 681,127 size 37x43; Picture "图形_29"

screen "系统画面" 800x480, template "Template_1"
   on GenerateScreen: SetTag("Tag_ScreenNumber", 3)
   Button "HmiScreenItemData" at 36,146 size 159x47; TextOff 'SIMATIC PLC 系统诊断'; PictureOff "Navigates to SIMATIC PLC 系统诊断 for KTP700 Basic+ PN 14.0.0.0"; PictureOn "Navigates to SIMATIC PLC 系统诊断 for KTP700 Basic+ PN 14.0.0.0"
      on Release: ActivateScreen("SIMATIC PLC 系统诊断", 0)
   Button "HmiScreenItemData_1" at 36,205 size 159x47; TextOff '用户管理'; PictureOff "Navigates to 用户管理 for KTP700 Basic+ PN 14.0.0.0"; PictureOn "Navigates to 用户管理 for KTP700 Basic+ PN 14.0.0.0"
      on Release: ActivateScreen("用户管理", 0)

screen "SIMATIC PLC 系统诊断" 800x480, template "Template_1"
   on GenerateScreen: SetTag("Tag_ScreenNumber", 4)
   SysDiagControl "HmiScreenItemData" at 1,50 size 796x371

screen "用户管理" 800x480, template "Template_1"
   on GenerateScreen: SetTag("Tag_ScreenNumber", 5)
   UserView "HmiScreenItemData" at 1,49 size 796x372

screen "趋势" 800x480, template "Template_1"
   on GenerateScreen: SetTag("Tag_ScreenNumber", 2)
   TextField "HmiScreenItemData" at 80,228 size 640x25; Text '画面 0'
   TrendView "趋势视图_1" at 1,49 size 798x377

screen "报警" 800x480, template "Template_1"
   on GenerateScreen: SetTag("Tag_ScreenNumber", 2)
   AlarmView "报警视图_1" at 1,49 size 798x375; AlarmLog "Alarm_log_1"

screen "参数配置" 800x480, template "Template_1"
   on GenerateScreen: SetTag("Tag_ScreenNumber", 2)
   Button "Template_Button_1" at 16,358 size 105x50; TextOff '运行时间清零 / ClearRuntime'; Authorization "User administration"
      on Press: SetBit("PARAM_CONFIG_DB_BT_Function_BT_Runtime_Reset")
      on Release: ResetBit("PARAM_CONFIG_DB_BT_Function_BT_Runtime_Reset")
   GraphicView "图形视图_1" at 24,50 size 84x75; Picture "图形_22"
   TextField "文本域_1" at 166,54 size 52x23; Text '名称 / Name'
   TextField "文本域_2" at 276,54 size 74x23; Text '设定值 / Setpoint'
   TextField "文本域_3" at 381,54 size 92x23; Text '初始值 / InitialVAL:'
   TextField "文本域_7" at 134,99 size 123x20; Text '主加热温度上限： / MainHeaterUpper:'
   TextField "文本域_8" at 134,127 size 117x20; Text '主加热温度下限： / MainHeaterFloor:'
   TextField "文本域_11" at 134,156 size 135x20; Text '加热超温报警温度: / HeatTemUpperLimit:'
   TextField "文本域_13" at 134,184 size 139x20; Text '露点超限温度： / DewPointUpperLimit:'
   TextField "文本域_14" at 134,213 size 97x20; Text '加热温度补偿: / HeatTemCom:'
   TextField "文本域_18" at 134,242 size 103x20; Text '压力温度补偿： / DewPointCom:'
   TextField "文本域_20" at 134,271 size 109x20; Text '工作露点设定: / DewpointUpper:'
   IOField "I/O 域_1" at 268,93 size 75x28; FormatPattern 99999
      ProcessValue <- "PARAM_CONFIG_DB_主加热温度上限"
   IOField "I/O 域_3" at 268,122 size 75x28; FormatPattern 99999
      ProcessValue <- "PARAM_CONFIG_DB_主加热温度下限"
   IOField "I/O 域_9" at 268,151 size 75x28; FormatPattern 99999
      ProcessValue <- "PARAM_CONFIG_DB_加热超限温度报警"
   IOField "I/O 域_13" at 268,180 size 75x28; FormatPattern s99999
      ProcessValue <- "PARAM_CONFIG_DB_露点超限温度"
   IOField "I/O 域_15" at 268,209 size 75x28; FormatPattern s99999
      ProcessValue <- "PARAM_CONFIG_DB_加热温度补偿"
   IOField "I/O 域_19" at 268,238 size 75x28; FormatPattern s99999
      ProcessValue <- "PARAM_CONFIG_DB_压力温度补偿"
   IOField "I/O 域_23" at 268,267 size 75x28; FormatPattern s99999
      ProcessValue <- "PARAM_CONFIG_DB_工作露点设定"
   TextField "文本域_4" at 370,93 size 78x28; Text '120℃'
   TextField "文本域_5" at 370,122 size 78x28; Text '100℃'
   TextField "文本域_16" at 370,151 size 78x28; Text '180℃'
   TextField "文本域_22" at 370,180 size 78x28; Text '-10℃'
   TextField "文本域_23" at 370,209 size 78x28; Text '0℃'
   TextField "文本域_25" at 370,238 size 78x28; Text '0℃'
   TextField "文本域_27" at 370,267 size 78x28; Text '-30℃'
   TextField "文本域_28" at 497,50 size 52x23; Text '名称 / Name'
   TextField "文本域_29" at 607,50 size 74x23; Text '设定值 / Setpoint'
   TextField "文本域_30" at 708,50 size 92x23; Text '初始值 / InitialVAL:'
   TextField "文本域_31" at 465,95 size 107x20; Text '停机充压时间： / PressurizeTime:'
   TextField "文本域_32" at 465,123 size 133x20; Text 'A塔工作B塔待再生： / B_Wait:'
   TextField "文本域_33" at 465,152 size 133x20; Text 'A塔工作B塔热再生： / B_Heat:'
   TextField "文本域_34" at 465,181 size 119x20; Text 'A塔工作B塔吹冷： / B_Cool:'
   TextField "文本域_35" at 465,210 size 119x20; Text 'A塔工作B塔充压： / B_Pressurize:'
   TextField "文本域_36" at 465,239 size 91x20; Text 'A塔B塔均压： / B_Balance:'
   TextField "文本域_37" at 465,267 size 103x20; Text '故障判断延时： / ErrorDelay:'
   TextField "文本域_38" at 465,296 size 103x20; Text '保养时间设定： / MaintainTime:'
   TextField "文本域_39" at 465,325 size 82x20; Text '从站地址： / SlaveADDR:'
   TextField "文本域_40" at 465,354 size 159x20; Text '露点控制最长延时： / DewPointLongestDealy:'
   IOField "I/O 域_2" at 599,89 size 75x28; FormatPattern 99999
      ProcessValue <- "PARAM_CONFIG_DB_停机充压时间"
   IOField "I/O 域_4" at 599,118 size 75x28; FormatPattern 99999
      ProcessValue <- "PARAM_CONFIG_DB_A塔工作B塔待再生"
   IOField "I/O 域_6" at 599,147 size 75x28; FormatPattern 99999
      ProcessValue <- "PARAM_CONFIG_DB_A塔工作B塔热再生"
   IOField "I/O 域_8" at 599,176 size 75x28; FormatPattern 99999
      ProcessValue <- "PARAM_CONFIG_DB_A塔工作B塔吹冷"
   IOField "I/O 域_10" at 599,205 size 75x28; FormatPattern 99999
      ProcessValue <- "PARAM_CONFIG_DB_A塔工作B塔充压"
   IOField "I/O 域_12" at 599,234 size 75x28; FormatPattern 99999
      ProcessValue <- "PARAM_CONFIG_DB_A塔B塔均压"
   IOField "I/O 域_14" at 599,263 size 75x28; FormatPattern 99999
      ProcessValue <- "PARAM_CONFIG_DB_故障判断延时"
   IOField "I/O 域_16" at 599,292 size 100x28; FormatPattern 9999999999
      ProcessValue <- "PARAM_CONFIG_DB_保养时间设定"
   IOField "I/O 域_18" at 599,321 size 75x28; FormatPattern 99999
      ProcessValue <- "PARAM_CONFIG_DB_从站地址"
   IOField "I/O 域_20" at 599,350 size 75x28; FormatPattern 99999
      ProcessValue <- "PARAM_CONFIG_DB_露点控制最长延时"
   TextField "文本域_43" at 701,89 size 78x28; Text '30秒 / 30s'
   TextField "文本域_44" at 701,118 size 78x28; Text '10秒 / 10s'
   TextField "文本域_45" at 701,147 size 78x28; Text '25分 / 25min'
   TextField "文本域_46" at 701,176 size 78x28; Text '15分 / 15min'
   TextField "文本域_47" at 701,205 size 78x28; Text '8分 / 8min'
   TextField "文本域_48" at 701,234 size 78x28; Text '10秒 / 10s'
   TextField "文本域_49" at 701,263 size 78x28; Text '5秒 / 10s'
   TextField "文本域_50" at 701,292 size 78x28; Text '0时 / 0'
   TextField "文本域_51" at 701,321 size 78x28; Text '2'
   TextField "文本域_52" at 701,350 size 78x28; Text '60分 / 60min'
   TextField "文本域_6" at 133,321 size 97x17; Text '保养倒记时间: / DewpointUpper:'
   IOField "I/O 域_5" at 265,314 size 100x28; FormatPattern s999999999
      ProcessValue <- "PARAM_CONFIG_DB_MaintainTime_CountdownValue"
   TextField "文本域_9" at 365,318 size 22x20; Text '时'
*)